	VAR jointtarget CDP_979 := [[-11.91, 35.75, 6.26, 0, 47.99, -88.67], [9E9, 9E9, 9E9, 9E9, 9E9, 9E9]];
	VAR jointtarget CDP_980 := [[-11.89, 35.75, 6.26, 0, 47.99, -88.98], [9E9, 9E9, 9E9, 9E9, 9E9, 9E9]];
	VAR jointtarget CDP_981 := [[-11.87, 35.75, 6.26, 0, 47.99, -89.63], [9E9, 9E9, 9E9, 9E9, 9E9, 9E9]];
	VAR jointtarget CDP_982 := [[-11.86, 35.75, 6.26, 0, 47.99, -90.27], [9E9, 9E9, 9E9, 9E9, 9E9, 9E9]];
	VAR jointtarget CDP_983 := [[-11.84, 35.75, 6.26, 0, 47.99, -90.92], [9E9, 9E9, 9E9, 9E9, 9E9, 9E9]];
	VAR jointtarget CDP_984 := [[-11.82, 35.75, 6.26, 0, 47.99, -91.56], [9E9, 9E9, 9E9, 9E9, 9E9, 9E9]];
	VAR jointtarget CDP_985 := [[-11.81, 35.75, 6.26, 0, 47.99, -92.21], [9E9, 9E9, 9E9, 9E9, 9E9, 9E9]];
	VAR jointtarget CDP_986 := [[-11.79, 35.75, 6.26, 0, 47.99, -92.85], [9E9, 9E9, 9E9, 9E9, 9E9, 9E9]];
	VAR jointtarget CDP_987 := [[-11.77, 35.75, 6.26, 0, 47.99, -93.5], [9E9, 9E9, 9E9, 9E9, 9E9, 9E9]];
	VAR jointtarget CDP_988 := [[-11.76, 35.75, 6.27, 0, 47.99, -94.14], [9E9, 9E9, 9E9, 9E9, 9E9, 9E9]];
	VAR jointtarget CDP_989 := [[-11.74, 35.74, 6.27, 0, 47.99, -94.79], [9E9, 9E9, 9E9, 9E9, 9E9, 9E9]];
	VAR jointtarget CDP_990 := [[-11.72, 35.74, 6.27, 0, 47.99, -95.43], [9E9, 9E9, 9E9, 9E9, 9E9, 9E9]];
	VAR jointtarget CDP_991 := [[-11.71, 35.74, 6.28, 0, 47.98, -96.08], [9E9, 9E9, 9E9, 9E9, 9E9, 9E9]];
	VAR jointtarget CDP_992 := [[-11.69, 35.74, 6.28, 0, 47.98, -96.72], [9E9, 9E9, 9E9, 9E9, 9E9, 9E9]];
	VAR jointtarget CDP_993 := [[-11.67, 35.74, 6.28, 0, 47.98, -97.37], [9E9, 9E9, 9E9, 9E9, 9E9, 9E9]];
	VAR jointtarget CDP_994 := [[-11.66, 35.73, 6.29, 0, 47.98, -98.01], [9E9, 9E9, 9E9, 9E9, 9E9, 9E9]];
	VAR jointtarget CDP_995 := [[-11.64, 35.73, 6.29, 0, 47.98, -98.66], [9E9, 9E9, 9E9, 9E9, 9E9, 9E9]];
	VAR jointtarget CDP_996 := [[-11.62, 35.73, 6.3, 0, 47.98, -99.31], [9E9, 9E9, 9E9, 9E9, 9E9, 9E9]];
	VAR jointtarget CDP_997 := [[-11.61, 35.72, 6.3, 0, 47.97, -99.95], [9E9, 9E9, 9E9, 9E9, 9E9, 9E9]];
	VAR jointtarget CDP_998 := [[-11.59, 35.72, 6.31, 0, 47.97, -100.6], [9E9, 9E9, 9E9, 9E9, 9E9, 9E9]];
	VAR jointtarget CDP_999 := [[-11.57, 35.72, 6.31, 0, 47.97, -101.24], [9E9, 9E9, 9E9, 9E9, 9E9, 9E9]];
	VAR jointtarget CDP_1000 := [[-10.48, 35.49, 6.71, 0, 47.81, -100.48], [9E9, 9E9, 9E9, 9E9, 9E9, 9E9]];
	VAR jointtarget CDP_1001 := [[-9.38, 35.28, 7.06, 0, 47.66, -99.38], [9E9, 9E9, 9E9, 9E9, 9E9, 9E9]];
	VAR jointtarget CDP_1002 := [[-8.27, 35.1, 7.37, 0, 47.53, -98.27], [9E9, 9E9, 9E9, 9E9, 9E9, 9E9]];
	VAR jointtarget CDP_1003 := [[-7.15, 34.94, 7.64, 0, 47.42, -97.15], [9E9, 9E9, 9E9, 9E9, 9E9, 9E9]];
	VAR jointtarget CDP_1004 := [[-6.03, 34.8, 7.88, 0, 47.32, -96.03], [9E9, 9E9, 9E9, 9E9, 9E9, 9E9]];
	VAR jointtarget CDP_1005 := [[-4.9, 34.69, 8.07, 0, 47.24, -94.9], [9E9, 9E9, 9E9, 9E9, 9E9, 9E9]];
	VAR jointtarget CDP_1006 := [[-3.77, 34.6, 8.22, 0, 47.18, -93.77], [9E9, 9E9, 9E9, 9E9, 9E9, 9E9]];
	VAR jointtarget CDP_1007 := [[-2.64, 34.53, 8.33, 0, 47.13, -92.64], [9E9, 9E9, 9E9, 9E9, 9E9, 9E9]];
	VAR jointtarget CDP_1008 := [[-1.51, 34.49, 8.41, 0, 47.1, -91.51], [9E9, 9E9, 9E9, 9E9, 9E9, 9E9]];
	VAR jointtarget CDP_1009 := [[-0.37, 34.47, 8.44, 0, 47.09, -90.37], [9E9, 9E9, 9E9, 9E9, 9E9, 9E9]];
	VAR jointtarget CDP_1010 := [[0.76, 34.48, 8.43, 0, 47.09, -89.24], [9E9, 9E9, 9E9, 9E9, 9E9, 9E9]];
	VAR jointtarget CDP_1011 := [[1.9, 34.5, 8.39, 0, 47.11, -88.1], [9E9, 9E9, 9E9, 9E9, 9E9, 9E9]];
	VAR jointtarget CDP_1012 := [[3.03, 34.55, 8.3, 0, 47.15, -86.97], [9E9, 9E9, 9E9, 9E9, 9E9, 9E9]];
	VAR jointtarget CDP_1013 := [[4.16, 34.63, 8.17, 0, 47.2, -85.84], [9E9, 9E9, 9E9, 9E9, 9E9, 9E9]];
	VAR jointtarget CDP_1014 := [[5.29, 34.73, 8.01, 0, 47.27, -84.71], [9E9, 9E9, 9E9, 9E9, 9E9, 9E9]];
	VAR jointtarget CDP_1015 := [[6.42, 34.85, 7.8, 0, 47.35, -83.58], [9E9, 9E9, 9E9, 9E9, 9E9, 9E9]];
	VAR jointtarget CDP_1016 := [[7.54, 34.99, 7.55, 0, 47.45, -82.46], [9E9, 9E9, 9E9, 9E9, 9E9, 9E9]];
	VAR jointtarget CDP_1017 := [[8.65, 35.16, 7.27, 0, 47.57, -81.35], [9E9, 9E9, 9E9, 9E9, 9E9, 9E9]];
	VAR jointtarget CDP_1018 := [[9.76, 35.35, 6.94, 0, 47.71, -80.24], [9E9, 9E9, 9E9, 9E9, 9E9, 9E9]];
	VAR jointtarget CDP_1019 := [[10.86, 35.56, 6.58, 0, 47.86, -79.14], [9E9, 9E9, 9E9, 9E9, 9E9, 9E9]];
	VAR jointtarget CDP_1020 := [[10.87, 35.57, 6.57, 0, 47.86, -79.46], [9E9, 9E9, 9E9, 9E9, 9E9, 9E9]];
	VAR jointtarget CDP_1021 := [[10.89, 35.57, 6.56, 0, 47.86, -80.1], [9E9, 9E9, 9E9, 9E9, 9E9, 9E9]];
	VAR jointtarget CDP_1022 := [[10.91, 35.57, 6.56, 0, 47.87, -80.75], [9E9, 9E9, 9E9, 9E9, 9E9, 9E9]];
	VAR jointtarget CDP_1023 := [[10.92, 35.58, 6.55, 0, 47.87, -81.39], [9E9, 9E9, 9E9, 9E9, 9E9, 9E9]];
	VAR jointtarget CDP_1024 := [[10.94, 35.58, 6.55, 0, 47.87, -82.04], [9E9, 9E9, 9E9, 9E9, 9E9, 9E9]];
	VAR jointtarget CDP_1025 := [[10.96, 35.58, 6.55, 0, 47.87, -82.68], [9E9, 9E9, 9E9, 9E9, 9E9, 9E9]];
	VAR jointtarget CDP_1026 := [[10.97, 35.58, 6.54, 0, 47.87, -83.33], [9E9, 9E9, 9E9, 9E9, 9E9, 9E9]];
	VAR jointtarget CDP_1027 := [[10.99, 35.59, 6.54, 0, 47.87, -83.97], [9E9, 9E9, 9E9, 9E9, 9E9, 9E9]];
	VAR jointtarget CDP_1028 := [[11.01, 35.59, 6.54, 0, 47.88, -84.62], [9E9, 9E9, 9E9, 9E9, 9E9, 9E9]];
	VAR jointtarget CDP_1029 := [[11.02, 35.59, 6.53, 0, 47.88, -85.27], [9E9, 9E9, 9E9, 9E9, 9E9, 9E9]];
	VAR jointtarget CDP_1030 := [[11.04, 35.59, 6.53, 0, 47.88, -85.91], [9E9, 9E9, 9E9, 9E9, 9E9, 9E9]];
	VAR jointtarget CDP_1031 := [[11.06, 35.59, 6.53, 0, 47.88, -86.56], [9E9, 9E9, 9E9, 9E9, 9E9, 9E9]];
	VAR jointtarget CDP_1032 := [[11.07, 35.59, 6.53, 0, 47.88, -87.2], [9E9, 9E9, 9E9, 9E9, 9E9, 9E9]];
	VAR jointtarget CDP_1033 := [[11.09, 35.59, 6.53, 0, 47.88, -87.85], [9E9, 9E9, 9E9, 9E9, 9E9, 9E9]];
	VAR jointtarget CDP_1034 := [[11.11, 35.59, 6.53, 0, 47.88, -88.49], [9E9, 9E9, 9E9, 9E9, 9E9, 9E9]];
	VAR jointtarget CDP_1035 := [[11.13, 35.59, 6.53, 0, 47.88, -89.14], [9E9, 9E9, 9E9, 9E9, 9E9, 9E9]];
	VAR jointtarget CDP_1036 := [[11.14, 35.59, 6.53, 0, 47.88, -89.78], [9E9, 9E9, 9E9, 9E9, 9E9, 9E9]];
	VAR jointtarget CDP_1037 := [[11.16, 35.59, 6.53, 0, 47.88, -90.43], [9E9, 9E9, 9E9, 9E9, 9E9, 9E9]];
	VAR jointtarget CDP_1038 := [[11.18, 35.59, 6.53, 0, 47.88, -91.07], [9E9, 9E9, 9E9, 9E9, 9E9, 9E9]];
	VAR jointtarget CDP_1039 := [[11.19, 35.59, 6.53, 0, 47.88, -91.72], [9E9, 9E9, 9E9, 9E9, 9E9, 9E9]];
	VAR jointtarget CDP_1040 := [[11.26, 35.59, 6.53, 0, 47.88, -91.98], [9E9, 9E9, 9E9, 9E9, 9E9, 9E9]];
	VAR jointtarget CDP_1041 := [[11.33, 35.59, 6.54, 0, 47.88, -91.91], [9E9, 9E9, 9E9, 9E9, 9E9, 9E9]];
	VAR jointtarget CDP_1042 := [[11.4, 35.59, 6.54, 0, 47.87, -91.84], [9E9, 9E9, 9E9, 9E9, 9E9, 9E9]];
	VAR jointtarget CDP_1043 := [[11.47, 35.58, 6.54, 0, 47.87, -91.78], [9E9, 9E9, 9E9, 9E9, 9E9, 9E9]];
	VAR jointtarget CDP_1044 := [[11.53, 35.58, 6.55, 0, 47.87, -91.71], [9E9, 9E9, 9E9, 9E9, 9E9, 9E9]];
	VAR jointtarget CDP_1045 := [[11.6, 35.58, 6.55, 0, 47.87, -91.64], [9E9, 9E9, 9E9, 9E9, 9E9, 9E9]];
	VAR jointtarget CDP_1046 := [[11.67, 35.58, 6.56, 0, 47.87, -91.57], [9E9, 9E9, 9E9, 9E9, 9E9, 9E9]];
	VAR jointtarget CDP_1047 := [[11.74, 35.57, 6.56, 0, 47.87, -91.5], [9E9, 9E9, 9E9, 9E9, 9E9, 9E9]];
	VAR jointtarget CDP_1048 := [[11.81, 35.57, 6.56, 0, 47.87, -91.44], [9E9, 9E9, 9E9, 9E9, 9E9, 9E9]];
	VAR jointtarget CDP_1049 := [[11.87, 35.57, 6.56, 0, 47.86, -91.37], [9E9, 9E9, 9E9, 9E9, 9E9, 9E9]];
	VAR jointtarget CDP_1050 := [[11.94, 35.57, 6.57, 0, 47.86, -91.3], [9E9, 9E9, 9E9, 9E9, 9E9, 9E9]];
	VAR jointtarget CDP_1051 := [[12.01, 35.57, 6.57, 0, 47.86, -91.23], [9E9, 9E9, 9E9, 9E9, 9E9, 9E9]];
	VAR jointtarget CDP_1052 := [[12.08, 35.57, 6.57, 0, 47.86, -91.16], [9E9, 9E9, 9E9, 9E9, 9E9, 9E9]];
	VAR jointtarget CDP_1053 := [[12.15, 35.56, 6.58, 0, 47.86, -91.09], [9E9, 9E9, 9E9, 9E9, 9E9, 9E9]];
	VAR jointtarget CDP_1054 := [[12.21, 35.56, 6.58, 0, 47.86, -91.03], [9E9, 9E9, 9E9, 9E9, 9E9, 9E9]];
	VAR jointtarget CDP_1055 := [[12.28, 35.56, 6.58, 0, 47.86, -90.96], [9E9, 9E9, 9E9, 9E9, 9E9, 9E9]];
	VAR jointtarget CDP_1056 := [[12.35, 35.56, 6.58, 0, 47.86, -90.89], [9E9, 9E9, 9E9, 9E9, 9E9, 9E9]];
	VAR jointtarget CDP_1057 := [[12.42, 35.56, 6.58, 0, 47.86, -90.82], [9E9, 9E9, 9E9, 9E9, 9E9, 9E9]];
	VAR jointtarget CDP_1058 := [[12.49, 35.56, 6.59, 0, 47.86, -90.75], [9E9, 9E9, 9E9, 9E9, 9E9, 9E9]];
	VAR jointtarget CDP_1059 := [[12.55, 35.56, 6.59, 0, 47.86, -90.69], [9E9, 9E9, 9E9, 9E9, 9E9, 9E9]];
	VAR jointtarget CDP_1060 := [[12.69, 35.57, 6.57, 0, 47.86, -85.39], [9E9, 9E9, 9E9, 9E9, 9E9, 9E9]];
	VAR jointtarget CDP_1061 := [[12.81, 35.61, 6.51, 0, 47.89, -74.94], [9E9, 9E9, 9E9, 9E9, 9E9, 9E9]];
	VAR jointtarget CDP_1062 := [[12.93, 35.67, 6.4, 0, 47.93, -64.5], [9E9, 9E9, 9E9, 9E9, 9E9, 9E9]];
	VAR jointtarget CDP_1063 := [[13.04, 35.75, 6.26, 0, 47.99, -54.07], [9E9, 9E9, 9E9, 9E9, 9E9, 9E9]];
	VAR jointtarget CDP_1064 := [[13.13, 35.85, 6.08, 0, 48.07, -43.65], [9E9, 9E9, 9E9, 9E9, 9E9, 9E9]];
	VAR jointtarget CDP_1065 := [[13.2, 35.97, 5.88, 0, 48.15, -33.25], [9E9, 9E9, 9E9, 9E9, 9E9, 9E9]];
	VAR jointtarget CDP_1066 := [[13.25, 36.1, 5.65, 0, 48.24, -22.88], [9E9, 9E9, 9E9, 9E9, 9E9, 9E9]];
	VAR jointtarget CDP_1067 := [[13.28, 36.24, 5.41, 0, 48.34, -12.53], [9E9, 9E9, 9E9, 9E9, 9E9, 9E9]];
	VAR jointtarget CDP_1068 := [[13.29, 36.39, 5.17, 0, 48.45, -2.2], [9E9, 9E9, 9E9, 9E9, 9E9, 9E9]];
	VAR jointtarget CDP_1069 := [[13.27, 36.53, 4.92, 0, 48.55, 8.11], [9E9, 9E9, 9E9, 9E9, 9E9, 9E9]];
	VAR jointtarget CDP_1070 := [[13.23, 36.66, 4.69, 0, 48.65, 18.39], [9E9, 9E9, 9E9, 9E9, 9E9, 9E9]];
	VAR jointtarget CDP_1071 := [[13.17, 36.79, 4.47, 0, 48.74, 28.65], [9E9, 9E9, 9E9, 9E9, 9E9, 9E9]];
	VAR jointtarget CDP_1072 := [[13.08, 36.9, 4.28, 0, 48.82, 38.9], [9E9, 9E9, 9E9, 9E9, 9E9, 9E9]];
	VAR jointtarget CDP_1073 := [[12.99, 36.99, 4.12, 0, 48.89, 49.12], [9E9, 9E9, 9E9, 9E9, 9E9, 9E9]];
	VAR jointtarget CDP_1074 := [[12.88, 37.07, 3.99, 0, 48.94, 59.33], [9E9, 9E9, 9E9, 9E9, 9E9, 9E9]];
	VAR jointtarget CDP_1075 := [[12.75, 37.12, 3.91, 0, 48.98, 69.54], [9E9, 9E9, 9E9, 9E9, 9E9, 9E9]];
	VAR jointtarget CDP_1076 := [[12.63, 37.14, 3.86, 0, 48.99, 79.73], [9E9, 9E9, 9E9, 9E9, 9E9, 9E9]];
	VAR jointtarget CDP_1077 := [[12.5, 37.14, 3.86, 0, 48.99, 89.93], [9E9, 9E9, 9E9, 9E9, 9E9, 9E9]];
	VAR jointtarget CDP_1078 := [[12.37, 37.12, 3.91, 0, 48.98, 100.13], [9E9, 9E9, 9E9, 9E9, 9E9, 9E9]];
	VAR jointtarget CDP_1079 := [[12.25, 37.07, 3.99, 0, 48.94, 110.33], [9E9, 9E9, 9E9, 9E9, 9E9, 9E9]];
	VAR jointtarget CDP_1080 := [[12.19, 37.04, 4.05, 0, 48.92, 115.43], [9E9, 9E9, 9E9, 9E9, 9E9, 9E9]];
	VAR jointtarget CDP_1081 := [[12.13, 37, 4.1, 0, 48.89, 115.37], [9E9, 9E9, 9E9, 9E9, 9E9, 9E9]];
	VAR jointtarget CDP_1082 := [[12.07, 36.97, 4.16, 0, 48.87, 115.31], [9E9, 9E9, 9E9, 9E9, 9E9, 9E9]];
	VAR jointtarget CDP_1083 := [[12.01, 36.94, 4.21, 0, 48.85, 115.25], [9E9, 9E9, 9E9, 9E9, 9E9, 9E9]];
	VAR jointtarget CDP_1084 := [[11.95, 36.91, 4.27, 0, 48.82, 115.19], [9E9, 9E9, 9E9, 9E9, 9E9, 9E9]];
	VAR jointtarget CDP_1085 := [[11.89, 36.88, 4.32, 0, 48.8, 115.13], [9E9, 9E9, 9E9, 9E9, 9E9, 9E9]];
	VAR jointtarget CDP_1086 := [[11.83, 36.85, 4.37, 0, 48.78, 115.07], [9E9, 9E9, 9E9, 9E9, 9E9, 9E9]];
	VAR jointtarget CDP_1087 := [[11.77, 36.82, 4.43, 0, 48.76, 115.01], [9E9, 9E9, 9E9, 9E9, 9E9, 9E9]];
	VAR jointtarget CDP_1088 := [[11.71, 36.78, 4.48, 0, 48.73, 114.95], [9E9, 9E9, 9E9, 9E9, 9E9, 9E9]];
	VAR jointtarget CDP_1089 := [[11.65, 36.75, 4.54, 0, 48.71, 114.89], [9E9, 9E9, 9E9, 9E9, 9E9, 9E9]];
	VAR jointtarget CDP_1090 := [[11.59, 36.72, 4.59, 0, 48.69, 114.83], [9E9, 9E9, 9E9, 9E9, 9E9, 9E9]];
	VAR jointtarget CDP_1091 := [[11.53, 36.69, 4.64, 0, 48.67, 114.77], [9E9, 9E9, 9E9, 9E9, 9E9, 9E9]];
	VAR jointtarget CDP_1092 := [[11.47, 36.66, 4.7, 0, 48.64, 114.71], [9E9, 9E9, 9E9, 9E9, 9E9, 9E9]];
	VAR jointtarget CDP_1093 := [[11.4, 36.63, 4.75, 0, 48.62, 114.64], [9E9, 9E9, 9E9, 9E9, 9E9, 9E9]];
	VAR jointtarget CDP_1094 := [[11.34, 36.6, 4.8, 0, 48.6, 114.58], [9E9, 9E9, 9E9, 9E9, 9E9, 9E9]];
	VAR jointtarget CDP_1095 := [[11.28, 36.57, 4.85, 0, 48.58, 114.52], [9E9, 9E9, 9E9, 9E9, 9E9, 9E9]];
	VAR jointtarget CDP_1096 := [[11.22, 36.54, 4.91, 0, 48.56, 114.46], [9E9, 9E9, 9E9, 9E9, 9E9, 9E9]];
	VAR jointtarget CDP_1097 := [[11.16, 36.51, 4.96, 0, 48.53, 114.4], [9E9, 9E9, 9E9, 9E9, 9E9, 9E9]];
	VAR jointtarget CDP_1098 := [[11.1, 36.48, 5.01, 0, 48.51, 114.34], [9E9, 9E9, 9E9, 9E9, 9E9, 9E9]];
	VAR jointtarget CDP_1099 := [[11.04, 36.45, 5.06, 0, 48.49, 114.28], [9E9, 9E9, 9E9, 9E9, 9E9, 9E9]];
	VAR jointtarget CDP_1100 := [[11.02, 36.44, 5.08, 0, 48.49, 113.93], [9E9, 9E9, 9E9, 9E9, 9E9, 9E9]];
	VAR jointtarget CDP_1101 := [[11.01, 36.43, 5.09, 0, 48.48, 113.26], [9E9, 9E9, 9E9, 9E9, 9E9, 9E9]];
	VAR jointtarget CDP_1102 := [[10.99, 36.43, 5.1, 0, 48.47, 112.58], [9E9, 9E9, 9E9, 9E9, 9E9, 9E9]];
	VAR jointtarget CDP_1103 := [[10.98, 36.42, 5.11, 0, 48.47, 111.9], [9E9, 9E9, 9E9, 9E9, 9E9, 9E9]];
	VAR jointtarget CDP_1104 := [[10.96, 36.41, 5.12, 0, 48.47, 111.22], [9E9, 9E9, 9E9, 9E9, 9E9, 9E9]];
	VAR jointtarget CDP_1105 := [[10.95, 36.41, 5.13, 0, 48.46, 110.55], [9E9, 9E9, 9E9, 9E9, 9E9, 9E9]];
	VAR jointtarget CDP_1106 := [[10.93, 36.4, 5.14, 0, 48.46, 109.87], [9E9, 9E9, 9E9, 9E9, 9E9, 9E9]];
	VAR jointtarget CDP_1107 := [[10.91, 36.39, 5.16, 0, 48.45, 109.19], [9E9, 9E9, 9E9, 9E9, 9E9, 9E9]];
	VAR jointtarget CDP_1108 := [[10.9, 36.39, 5.17, 0, 48.45, 108.51], [9E9, 9E9, 9E9, 9E9, 9E9, 9E9]];
	VAR jointtarget CDP_1109 := [[10.88, 36.38, 5.17, 0, 48.44, 107.83], [9E9, 9E9, 9E9, 9E9, 9E9, 9E9]];
	VAR jointtarget CDP_1110 := [[10.87, 36.38, 5.18, 0, 48.44, 107.16], [9E9, 9E9, 9E9, 9E9, 9E9, 9E9]];
	VAR jointtarget CDP_1111 := [[10.85, 36.37, 5.19, 0, 48.44, 106.48], [9E9, 9E9, 9E9, 9E9, 9E9, 9E9]];
	VAR jointtarget CDP_1112 := [[10.83, 36.37, 5.2, 0, 48.43, 105.8], [9E9, 9E9, 9E9, 9E9, 9E9, 9E9]];
	VAR jointtarget CDP_1113 := [[10.82, 36.36, 5.21, 0, 48.43, 105.12], [9E9, 9E9, 9E9, 9E9, 9E9, 9E9]];
	VAR jointtarget CDP_1114 := [[10.8, 36.36, 5.22, 0, 48.43, 104.44], [9E9, 9E9, 9E9, 9E9, 9E9, 9E9]];
	VAR jointtarget CDP_1115 := [[10.79, 36.35, 5.22, 0, 48.42, 103.77], [9E9, 9E9, 9E9, 9E9, 9E9, 9E9]];
	VAR jointtarget CDP_1116 := [[10.77, 36.35, 5.23, 0, 48.42, 103.09], [9E9, 9E9, 9E9, 9E9, 9E9, 9E9]];
	VAR jointtarget CDP_1117 := [[10.75, 36.34, 5.24, 0, 48.42, 102.41], [9E9, 9E9, 9E9, 9E9, 9E9, 9E9]];
	VAR jointtarget CDP_1118 := [[10.74, 36.34, 5.24, 0, 48.41, 101.73], [9E9, 9E9, 9E9, 9E9, 9E9, 9E9]];
	VAR jointtarget CDP_1119 := [[10.72, 36.34, 5.25, 0, 48.41, 101.05], [9E9, 9E9, 9E9, 9E9, 9E9, 9E9]];
	VAR jointtarget CDP_1120 := [[9.64, 36.13, 5.61, 0, 48.26, 99.64], [9E9, 9E9, 9E9, 9E9, 9E9, 9E9]];
	VAR jointtarget CDP_1121 := [[8.56, 35.94, 5.94, 0, 48.13, 98.56], [9E9, 9E9, 9E9, 9E9, 9E9, 9E9]];
	VAR jointtarget CDP_1122 := [[7.47, 35.77, 6.22, 0, 48.01, 97.47], [9E9, 9E9, 9E9, 9E9, 9E9, 9E9]];
	VAR jointtarget CDP_1123 := [[6.38, 35.63, 6.46, 0, 47.91, 96.38], [9E9, 9E9, 9E9, 9E9, 9E9, 9E9]];
	VAR jointtarget CDP_1124 := [[5.28, 35.51, 6.67, 0, 47.82, 95.28], [9E9, 9E9, 9E9, 9E9, 9E9, 9E9]];
	VAR jointtarget CDP_1125 := [[4.17, 35.41, 6.84, 0, 47.75, 94.17], [9E9, 9E9, 9E9, 9E9, 9E9, 9E9]];
	VAR jointtarget CDP_1126 := [[3.07, 35.34, 6.97, 0, 47.7, 93.07], [9E9, 9E9, 9E9, 9E9, 9E9, 9E9]];
	VAR jointtarget CDP_1127 := [[1.96, 35.28, 7.05, 0, 47.66, 91.96], [9E9, 9E9, 9E9, 9E9, 9E9, 9E9]];
	VAR jointtarget CDP_1128 := [[0.85, 35.26, 7.1, 0, 47.64, 90.85], [9E9, 9E9, 9E9, 9E9, 9E9, 9E9]];
	VAR jointtarget CDP_1129 := [[-0.26, 35.25, 7.11, 0, 47.64, 89.74], [9E9, 9E9, 9E9, 9E9, 9E9, 9E9]];
	VAR jointtarget CDP_1130 := [[-1.37, 35.27, 7.08, 0, 47.65, 88.63], [9E9, 9E9, 9E9, 9E9, 9E9, 9E9]];
	VAR jointtarget CDP_1131 := [[-2.48, 35.31, 7.02, 0, 47.68, 87.52], [9E9, 9E9, 9E9, 9E9, 9E9, 9E9]];
	VAR jointtarget CDP_1132 := [[-3.59, 35.37, 6.91, 0, 47.72, 86.41], [9E9, 9E9, 9E9, 9E9, 9E9, 9E9]];
	VAR jointtarget CDP_1133 := [[-4.7, 35.45, 6.76, 0, 47.78, 85.3], [9E9, 9E9, 9E9, 9E9, 9E9, 9E9]];
	VAR jointtarget CDP_1134 := [[-5.8, 35.56, 6.58, 0, 47.86, 84.2], [9E9, 9E9, 9E9, 9E9, 9E9, 9E9]];
	VAR jointtarget CDP_1135 := [[-6.9, 35.69, 6.35, 0, 47.95, 83.1], [9E9, 9E9, 9E9, 9E9, 9E9, 9E9]];
	VAR jointtarget CDP_1136 := [[-7.99, 35.85, 6.09, 0, 48.06, 82.01], [9E9, 9E9, 9E9, 9E9, 9E9, 9E9]];
	VAR jointtarget CDP_1137 := [[-9.08, 36.02, 5.79, 0, 48.19, 80.92], [9E9, 9E9, 9E9, 9E9, 9E9, 9E9]];
	VAR jointtarget CDP_1138 := [[-10.16, 36.22, 5.45, 0, 48.33, 79.84], [9E9, 9E9, 9E9, 9E9, 9E9, 9E9]];
	VAR jointtarget CDP_1139 := [[-11.23, 36.45, 5.07, 0, 48.49, 78.77], [9E9, 9E9, 9E9, 9E9, 9E9, 9E9]];
	VAR jointtarget CDP_1140 := [[-11.28, 36.46, 5.05, 0, 48.5, 79.81], [9E9, 9E9, 9E9, 9E9, 9E9, 9E9]];
	VAR jointtarget CDP_1141 := [[-11.34, 36.46, 5.03, 0, 48.5, 81.95], [9E9, 9E9, 9E9, 9E9, 9E9, 9E9]];
	VAR jointtarget CDP_1142 := [[-11.39, 36.47, 5.02, 0, 48.51, 84.09], [9E9, 9E9, 9E9, 9E9, 9E9, 9E9]];
	VAR jointtarget CDP_1143 := [[-11.45, 36.47, 5.02, 0, 48.51, 86.23], [9E9, 9E9, 9E9, 9E9, 9E9, 9E9]];
	VAR jointtarget CDP_1144 := [[-11.5, 36.48, 5.01, 0, 48.51, 88.37], [9E9, 9E9, 9E9, 9E9, 9E9, 9E9]];
	VAR jointtarget CDP_1145 := [[-11.56, 36.48, 5.01, 0, 48.51, 90.51], [9E9, 9E9, 9E9, 9E9, 9E9, 9E9]];
	VAR jointtarget CDP_1146 := [[-11.61, 36.47, 5.02, 0, 48.51, 92.65], [9E9, 9E9, 9E9, 9E9, 9E9, 9E9]];
	VAR jointtarget CDP_1147 := [[-11.67, 36.47, 5.03, 0, 48.51, 94.78], [9E9, 9E9, 9E9, 9E9, 9E9, 9E9]];
	VAR jointtarget CDP_1148 := [[-11.72, 36.46, 5.04, 0, 48.5, 96.92], [9E9, 9E9, 9E9, 9E9, 9E9, 9E9]];
	VAR jointtarget CDP_1149 := [[-11.78, 36.45, 5.06, 0, 48.49, 99.06], [9E9, 9E9, 9E9, 9E9, 9E9, 9E9]];
	VAR jointtarget CDP_1150 := [[-11.83, 36.44, 5.08, 0, 48.48, 101.2], [9E9, 9E9, 9E9, 9E9, 9E9, 9E9]];
	VAR jointtarget CDP_1151 := [[-11.89, 36.43, 5.1, 0, 48.47, 103.34], [9E9, 9E9, 9E9, 9E9, 9E9, 9E9]];
	VAR jointtarget CDP_1152 := [[-11.94, 36.41, 5.13, 0, 48.46, 105.48], [9E9, 9E9, 9E9, 9E9, 9E9, 9E9]];
	VAR jointtarget CDP_1153 := [[-11.99, 36.39, 5.16, 0, 48.45, 107.63], [9E9, 9E9, 9E9, 9E9, 9E9, 9E9]];
	VAR jointtarget CDP_1154 := [[-12.04, 36.37, 5.19, 0, 48.44, 109.77], [9E9, 9E9, 9E9, 9E9, 9E9, 9E9]];
	VAR jointtarget CDP_1155 := [[-12.09, 36.35, 5.23, 0, 48.42, 111.91], [9E9, 9E9, 9E9, 9E9, 9E9, 9E9]];
	VAR jointtarget CDP_1156 := [[-12.15, 36.32, 5.28, 0, 48.4, 114.05], [9E9, 9E9, 9E9, 9E9, 9E9, 9E9]];
	VAR jointtarget CDP_1157 := [[-12.19, 36.3, 5.32, 0, 48.38, 116.2], [9E9, 9E9, 9E9, 9E9, 9E9, 9E9]];
	VAR jointtarget CDP_1158 := [[-12.24, 36.27, 5.37, 0, 48.36, 118.34], [9E9, 9E9, 9E9, 9E9, 9E9, 9E9]];
	VAR jointtarget CDP_1159 := [[-12.29, 36.24, 5.42, 0, 48.34, 120.49], [9E9, 9E9, 9E9, 9E9, 9E9, 9E9]];
	VAR jointtarget CDP_1160 := [[-12.32, 36.22, 5.46, 0, 48.33, 121.56], [9E9, 9E9, 9E9, 9E9, 9E9, 9E9]];
	VAR jointtarget CDP_1161 := [[-12.35, 36.2, 5.49, 0, 48.31, 121.53], [9E9, 9E9, 9E9, 9E9, 9E9, 9E9]];
	VAR jointtarget CDP_1162 := [[-12.38, 36.18, 5.52, 0, 48.3, 121.5], [9E9, 9E9, 9E9, 9E9, 9E9, 9E9]];
	VAR jointtarget CDP_1163 := [[-12.41, 36.16, 5.55, 0, 48.29, 121.47], [9E9, 9E9, 9E9, 9E9, 9E9, 9E9]];
	VAR jointtarget CDP_1164 := [[-12.43, 36.14, 5.59, 0, 48.27, 121.44], [9E9, 9E9, 9E9, 9E9, 9E9, 9E9]];
	VAR jointtarget CDP_1165 := [[-12.46, 36.12, 5.62, 0, 48.26, 121.41], [9E9, 9E9, 9E9, 9E9, 9E9, 9E9]];
	VAR jointtarget CDP_1166 := [[-12.49, 36.1, 5.65, 0, 48.24, 121.39], [9E9, 9E9, 9E9, 9E9, 9E9, 9E9]];
	VAR jointtarget CDP_1167 := [[-12.52, 36.08, 5.68, 0, 48.23, 121.36], [9E9, 9E9, 9E9, 9E9, 9E9, 9E9]];
	VAR jointtarget CDP_1168 := [[-12.55, 36.07, 5.72, 0, 48.22, 121.33], [9E9, 9E9, 9E9, 9E9, 9E9, 9E9]];
	VAR jointtarget CDP_1169 := [[-12.58, 36.05, 5.75, 0, 48.2, 121.3], [9E9, 9E9, 9E9, 9E9, 9E9, 9E9]];
	VAR jointtarget CDP_1170 := [[-12.61, 36.03, 5.78, 0, 48.19, 121.27], [9E9, 9E9, 9E9, 9E9, 9E9, 9E9]];
	VAR jointtarget CDP_1171 := [[-12.63, 36.01, 5.81, 0, 48.18, 121.24], [9E9, 9E9, 9E9, 9E9, 9E9, 9E9]];
	VAR jointtarget CDP_1172 := [[-12.66, 35.99, 5.85, 0, 48.16, 121.21], [9E9, 9E9, 9E9, 9E9, 9E9, 9E9]];
	VAR jointtarget CDP_1173 := [[-12.69, 35.97, 5.88, 0, 48.15, 121.18], [9E9, 9E9, 9E9, 9E9, 9E9, 9E9]];
	VAR jointtarget CDP_1174 := [[-12.72, 35.95, 5.91, 0, 48.14, 121.16], [9E9, 9E9, 9E9, 9E9, 9E9, 9E9]];
	VAR jointtarget CDP_1175 := [[-12.75, 35.93, 5.94, 0, 48.12, 121.13], [9E9, 9E9, 9E9, 9E9, 9E9, 9E9]];
	VAR jointtarget CDP_1176 := [[-12.78, 35.91, 5.98, 0, 48.11, 121.1], [9E9, 9E9, 9E9, 9E9, 9E9, 9E9]];
	VAR jointtarget CDP_1177 := [[-12.81, 35.9, 6.01, 0, 48.1, 121.07], [9E9, 9E9, 9E9, 9E9, 9E9, 9E9]];
	VAR jointtarget CDP_1178 := [[-12.84, 35.88, 6.04, 0, 48.08, 121.04], [9E9, 9E9, 9E9, 9E9, 9E9, 9E9]];
	VAR jointtarget CDP_1179 := [[-12.86, 35.86, 6.07, 0, 48.07, 121.01], [9E9, 9E9, 9E9, 9E9, 9E9, 9E9]];
	VAR jointtarget CDP_1180 := [[-13.02, 35.79, 6.2, 0, 48.02, 114.17], [9E9, 9E9, 9E9, 9E9, 9E9, 9E9]];
	VAR jointtarget CDP_1181 := [[-13.18, 35.75, 6.25, 0, 47.99, 100.62], [9E9, 9E9, 9E9, 9E9, 9E9, 9E9]];
	VAR jointtarget CDP_1182 := [[-13.34, 35.76, 6.24, 0, 48, 87.07], [9E9, 9E9, 9E9, 9E9, 9E9, 9E9]];
	VAR jointtarget CDP_1183 := [[-13.5, 35.81, 6.15, 0, 48.04, 73.52], [9E9, 9E9, 9E9, 9E9, 9E9, 9E9]];
	VAR jointtarget CDP_1184 := [[-13.64, 35.9, 6, 0, 48.1, 59.99], [9E9, 9E9, 9E9, 9E9, 9E9, 9E9]];
	VAR jointtarget CDP_1185 := [[-13.76, 36.02, 5.79, 0, 48.19, 46.48], [9E9, 9E9, 9E9, 9E9, 9E9, 9E9]];
	VAR jointtarget CDP_1186 := [[-13.85, 36.17, 5.53, 0, 48.29, 33.01], [9E9, 9E9, 9E9, 9E9, 9E9, 9E9]];
	VAR jointtarget CDP_1187 := [[-13.91, 36.34, 5.25, 0, 48.41, 19.56], [9E9, 9E9, 9E9, 9E9, 9E9, 9E9]];
	VAR jointtarget CDP_1188 := [[-13.92, 36.52, 4.94, 0, 48.54, 6.16], [9E9, 9E9, 9E9, 9E9, 9E9, 9E9]];
	VAR jointtarget CDP_1189 := [[-13.9, 36.7, 4.63, 0, 48.67, -7.21], [9E9, 9E9, 9E9, 9E9, 9E9, 9E9]];
	VAR jointtarget CDP_1190 := [[-13.85, 36.86, 4.35, 0, 48.79, -20.54], [9E9, 9E9, 9E9, 9E9, 9E9, 9E9]];
	VAR jointtarget CDP_1191 := [[-13.76, 37.01, 4.09, 0, 48.9, -33.84], [9E9, 9E9, 9E9, 9E9, 9E9, 9E9]];
	VAR jointtarget CDP_1192 := [[-13.64, 37.13, 3.88, 0, 48.99, -47.11], [9E9, 9E9, 9E9, 9E9, 9E9, 9E9]];
	VAR jointtarget CDP_1193 := [[-13.5, 37.22, 3.72, 0, 49.05, -60.35], [9E9, 9E9, 9E9, 9E9, 9E9, 9E9]];
	VAR jointtarget CDP_1194 := [[-13.34, 37.27, 3.64, 0, 49.09, -73.59], [9E9, 9E9, 9E9, 9E9, 9E9, 9E9]];
	VAR jointtarget CDP_1195 := [[-13.18, 37.28, 3.62, 0, 49.1, -86.81], [9E9, 9E9, 9E9, 9E9, 9E9, 9E9]];
	VAR jointtarget CDP_1196 := [[-13.02, 37.25, 3.68, 0, 49.07, -100.04], [9E9, 9E9, 9E9, 9E9, 9E9, 9E9]];
	VAR jointtarget CDP_1197 := [[-12.88, 37.18, 3.8, 0, 49.02, -113.28], [9E9, 9E9, 9E9, 9E9, 9E9, 9E9]];
	VAR jointtarget CDP_1198 := [[-12.75, 37.07, 3.98, 0, 48.94, -126.54], [9E9, 9E9, 9E9, 9E9, 9E9, 9E9]];
	VAR jointtarget CDP_1199 := [[-12.64, 36.94, 4.22, 0, 48.84, -139.82], [9E9, 9E9, 9E9, 9E9, 9E9, 9E9]];
	VAR jointtarget CDP_1200 := [[-12.62, 36.89, 4.29, 0, 48.81, -146.49], [9E9, 9E9, 9E9, 9E9, 9E9, 9E9]];
	VAR jointtarget CDP_1201 := [[-12.59, 36.85, 4.36, 0, 48.78, -146.47], [9E9, 9E9, 9E9, 9E9, 9E9, 9E9]];
	VAR jointtarget CDP_1202 := [[-12.57, 36.81, 4.43, 0, 48.75, -146.44], [9E9, 9E9, 9E9, 9E9, 9E9, 9E9]];
	VAR jointtarget CDP_1203 := [[-12.54, 36.77, 4.5, 0, 48.72, -146.42], [9E9, 9E9, 9E9, 9E9, 9E9, 9E9]];
	VAR jointtarget CDP_1204 := [[-12.52, 36.73, 4.57, 0, 48.69, -146.4], [9E9, 9E9, 9E9, 9E9, 9E9, 9E9]];
	VAR jointtarget CDP_1205 := [[-12.49, 36.69, 4.65, 0, 48.67, -146.37], [9E9, 9E9, 9E9, 9E9, 9E9, 9E9]];
	VAR jointtarget CDP_1206 := [[-12.47, 36.65, 4.72, 0, 48.64, -146.35], [9E9, 9E9, 9E9, 9E9, 9E9, 9E9]];
	VAR jointtarget CDP_1207 := [[-12.44, 36.61, 4.79, 0, 48.61, -146.32], [9E9, 9E9, 9E9, 9E9, 9E9, 9E9]];
	VAR jointtarget CDP_1208 := [[-12.42, 36.57, 4.86, 0, 48.58, -146.3], [9E9, 9E9, 9E9, 9E9, 9E9, 9E9]];
	VAR jointtarget CDP_1209 := [[-12.39, 36.53, 4.93, 0, 48.55, -146.27], [9E9, 9E9, 9E9, 9E9, 9E9, 9E9]];
	VAR jointtarget CDP_1210 := [[-12.37, 36.48, 5, 0, 48.52, -146.25], [9E9, 9E9, 9E9, 9E9, 9E9, 9E9]];
	VAR jointtarget CDP_1211 := [[-12.34, 36.44, 5.07, 0, 48.49, -146.22], [9E9, 9E9, 9E9, 9E9, 9E9, 9E9]];
	VAR jointtarget CDP_1212 := [[-12.32, 36.4, 5.14, 0, 48.46, -146.2], [9E9, 9E9, 9E9, 9E9, 9E9, 9E9]];
	VAR jointtarget CDP_1213 := [[-12.29, 36.36, 5.21, 0, 48.43, -146.17], [9E9, 9E9, 9E9, 9E9, 9E9, 9E9]];
	VAR jointtarget CDP_1214 := [[-12.27, 36.32, 5.28, 0, 48.4, -146.15], [9E9, 9E9, 9E9, 9E9, 9E9, 9E9]];
	VAR jointtarget CDP_1215 := [[-12.24, 36.28, 5.35, 0, 48.37, -146.12], [9E9, 9E9, 9E9, 9E9, 9E9, 9E9]];
	VAR jointtarget CDP_1216 := [[-12.22, 36.24, 5.42, 0, 48.34, -146.1], [9E9, 9E9, 9E9, 9E9, 9E9, 9E9]];
	VAR jointtarget CDP_1217 := [[-12.19, 36.2, 5.49, 0, 48.31, -146.07], [9E9, 9E9, 9E9, 9E9, 9E9, 9E9]];
	VAR jointtarget CDP_1218 := [[-12.17, 36.16, 5.56, 0, 48.28, -146.05], [9E9, 9E9, 9E9, 9E9, 9E9, 9E9]];
	VAR jointtarget CDP_1219 := [[-12.14, 36.12, 5.63, 0, 48.25, -146.02], [9E9, 9E9, 9E9, 9E9, 9E9, 9E9]];
	VAR jointtarget CDP_1220 := [[-12.14, 36.1, 5.65, 0, 48.24, -145.46], [9E9, 9E9, 9E9, 9E9, 9E9, 9E9]];
	VAR jointtarget CDP_1221 := [[-12.13, 36.09, 5.67, 0, 48.24, -144.35], [9E9, 9E9, 9E9, 9E9, 9E9, 9E9]];
	VAR jointtarget CDP_1222 := [[-12.12, 36.08, 5.69, 0, 48.23, -143.24], [9E9, 9E9, 9E9, 9E9, 9E9, 9E9]];
	VAR jointtarget CDP_1223 := [[-12.11, 36.07, 5.71, 0, 48.22, -142.13], [9E9, 9E9, 9E9, 9E9, 9E9, 9E9]];
	VAR jointtarget CDP_1224 := [[-12.1, 36.06, 5.73, 0, 48.21, -141.01], [9E9, 9E9, 9E9, 9E9, 9E9, 9E9]];
	VAR jointtarget CDP_1225 := [[-12.09, 36.04, 5.75, 0, 48.2, -139.9], [9E9, 9E9, 9E9, 9E9, 9E9, 9E9]];
	VAR jointtarget CDP_1226 := [[-12.08, 36.03, 5.77, 0, 48.19, -138.79], [9E9, 9E9, 9E9, 9E9, 9E9, 9E9]];
	VAR jointtarget CDP_1227 := [[-12.07, 36.02, 5.79, 0, 48.19, -137.68], [9E9, 9E9, 9E9, 9E9, 9E9, 9E9]];
	VAR jointtarget CDP_1228 := [[-12.06, 36.01, 5.81, 0, 48.18, -136.56], [9E9, 9E9, 9E9, 9E9, 9E9, 9E9]];
	VAR jointtarget CDP_1229 := [[-12.05, 36, 5.83, 0, 48.17, -135.45], [9E9, 9E9, 9E9, 9E9, 9E9, 9E9]];
	VAR jointtarget CDP_1230 := [[-12.04, 35.99, 5.85, 0, 48.16, -134.34], [9E9, 9E9, 9E9, 9E9, 9E9, 9E9]];
	VAR jointtarget CDP_1231 := [[-12.03, 35.98, 5.87, 0, 48.16, -133.22], [9E9, 9E9, 9E9, 9E9, 9E9, 9E9]];
	VAR jointtarget CDP_1232 := [[-12.02, 35.97, 5.88, 0, 48.15, -132.11], [9E9, 9E9, 9E9, 9E9, 9E9, 9E9]];
	VAR jointtarget CDP_1233 := [[-12.01, 35.96, 5.9, 0, 48.14, -130.99], [9E9, 9E9, 9E9, 9E9, 9E9, 9E9]];
	VAR jointtarget CDP_1234 := [[-12, 35.95, 5.92, 0, 48.14, -129.88], [9E9, 9E9, 9E9, 9E9, 9E9, 9E9]];
	VAR jointtarget CDP_1235 := [[-11.99, 35.94, 5.93, 0, 48.13, -128.76], [9E9, 9E9, 9E9, 9E9, 9E9, 9E9]];
	VAR jointtarget CDP_1236 := [[-11.98, 35.93, 5.95, 0, 48.12, -127.65], [9E9, 9E9, 9E9, 9E9, 9E9, 9E9]];
	VAR jointtarget CDP_1237 := [[-11.97, 35.92, 5.97, 0, 48.12, -126.53], [9E9, 9E9, 9E9, 9E9, 9E9, 9E9]];
	VAR jointtarget CDP_1238 := [[-11.96, 35.91, 5.98, 0, 48.11, -125.42], [9E9, 9E9, 9E9, 9E9, 9E9, 9E9]];
	VAR jointtarget CDP_1239 := [[-11.95, 35.9, 5.99, 0, 48.11, -124.3], [9E9, 9E9, 9E9, 9E9, 9E9, 9E9]];
	VAR jointtarget CDP_1240 := [[-11.94, 35.89, 6.01, 0, 48.1, -123.74], [9E9, 9E9, 9E9, 9E9, 9E9, 9E9]];
	VAR jointtarget CDP_1241 := [[-11.93, 35.88, 6.02, 0, 48.1, -123.73], [9E9, 9E9, 9E9, 9E9, 9E9, 9E9]];
	VAR jointtarget CDP_1242 := [[-11.92, 35.87, 6.03, 0, 48.09, -123.72], [9E9, 9E9, 9E9, 9E9, 9E9, 9E9]];
	VAR jointtarget CDP_1243 := [[-11.9, 35.87, 6.05, 0, 48.09, -123.71], [9E9, 9E9, 9E9, 9E9, 9E9, 9E9]];
	VAR jointtarget CDP_1244 := [[-11.89, 35.86, 6.06, 0, 48.08, -123.7], [9E9, 9E9, 9E9, 9E9, 9E9, 9E9]];
	VAR jointtarget CDP_1245 := [[-11.88, 35.85, 6.07, 0, 48.08, -123.69], [9E9, 9E9, 9E9, 9E9, 9E9, 9E9]];
	VAR jointtarget CDP_1246 := [[-11.87, 35.84, 6.08, 0, 48.07, -123.68], [9E9, 9E9, 9E9, 9E9, 9E9, 9E9]];
	VAR jointtarget CDP_1247 := [[-11.86, 35.84, 6.1, 0, 48.07, -123.66], [9E9, 9E9, 9E9, 9E9, 9E9, 9E9]];
	VAR jointtarget CDP_1248 := [[-11.85, 35.83, 6.11, 0, 48.06, -123.65], [9E9, 9E9, 9E9, 9E9, 9E9, 9E9]];
	VAR jointtarget CDP_1249 := [[-11.84, 35.82, 6.12, 0, 48.06, -123.64], [9E9, 9E9, 9E9, 9E9, 9E9, 9E9]];
	VAR jointtarget CDP_1250 := [[-11.83, 35.81, 6.13, 0, 48.05, -123.63], [9E9, 9E9, 9E9, 9E9, 9E9, 9E9]];
	VAR jointtarget CDP_1251 := [[-11.82, 35.8, 6.15, 0, 48.05, -123.62], [9E9, 9E9, 9E9, 9E9, 9E9, 9E9]];
	VAR jointtarget CDP_1252 := [[-11.81, 35.8, 6.16, 0, 48.04, -123.61], [9E9, 9E9, 9E9, 9E9, 9E9, 9E9]];
	VAR jointtarget CDP_1253 := [[-11.8, 35.79, 6.17, 0, 48.04, -123.6], [9E9, 9E9, 9E9, 9E9, 9E9, 9E9]];
	VAR jointtarget CDP_1254 := [[-11.79, 35.78, 6.19, 0, 48.03, -123.59], [9E9, 9E9, 9E9, 9E9, 9E9, 9E9]];
	VAR jointtarget CDP_1255 := [[-11.78, 35.77, 6.2, 0, 48.03, -123.58], [9E9, 9E9, 9E9, 9E9, 9E9, 9E9]];
	VAR jointtarget CDP_1256 := [[-11.77, 35.76, 6.21, 0, 48.02, -123.57], [9E9, 9E9, 9E9, 9E9, 9E9, 9E9]];
	VAR jointtarget CDP_1257 := [[-11.76, 35.76, 6.22, 0, 48.02, -123.56], [9E9, 9E9, 9E9, 9E9, 9E9, 9E9]];
	VAR jointtarget CDP_1258 := [[-11.75, 35.75, 6.24, 0, 48.02, -123.55], [9E9, 9E9, 9E9, 9E9, 9E9, 9E9]];
	VAR jointtarget CDP_1259 := [[-11.74, 35.74, 6.25, 0, 48.01, -123.54], [9E9, 9E9, 9E9, 9E9, 9E9, 9E9]];
	VAR jointtarget CDP_1260 := [[-10.65, 35.51, 6.65, 0, 47.85, -100.65], [9E9, 9E9, 9E9, 9E9, 9E9, 9E9]];
	VAR jointtarget CDP_1261 := [[-9.55, 35.3, 7, 0, 47.7, -99.55], [9E9, 9E9, 9E9, 9E9, 9E9, 9E9]];
	VAR jointtarget CDP_1262 := [[-8.44, 35.11, 7.32, 0, 47.57, -98.44], [9E9, 9E9, 9E9, 9E9, 9E9, 9E9]];
	VAR jointtarget CDP_1263 := [[-7.33, 34.95, 7.6, 0, 47.45, -97.33], [9E9, 9E9, 9E9, 9E9, 9E9, 9E9]];
	VAR jointtarget CDP_1264 := [[-6.21, 34.81, 7.84, 0, 47.35, -96.21], [9E9, 9E9, 9E9, 9E9, 9E9, 9E9]];
	VAR jointtarget CDP_1265 := [[-5.09, 34.69, 8.04, 0, 47.27, -95.09], [9E9, 9E9, 9E9, 9E9, 9E9, 9E9]];
	VAR jointtarget CDP_1266 := [[-3.96, 34.6, 8.2, 0, 47.2, -93.96], [9E9, 9E9, 9E9, 9E9, 9E9, 9E9]];
	VAR jointtarget CDP_1267 := [[-2.83, 34.53, 8.32, 0, 47.15, -92.83], [9E9, 9E9, 9E9, 9E9, 9E9, 9E9]];
	VAR jointtarget CDP_1268 := [[-1.7, 34.48, 8.4, 0, 47.12, -91.7], [9E9, 9E9, 9E9, 9E9, 9E9, 9E9]];
	VAR jointtarget CDP_1269 := [[-0.56, 34.46, 8.44, 0, 47.11, -90.56], [9E9, 9E9, 9E9, 9E9, 9E9, 9E9]];
	VAR jointtarget CDP_1270 := [[0.57, 34.46, 8.44, 0, 47.11, -89.43], [9E9, 9E9, 9E9, 9E9, 9E9, 9E9]];
	VAR jointtarget CDP_1271 := [[1.7, 34.48, 8.4, 0, 47.12, -88.3], [9E9, 9E9, 9E9, 9E9, 9E9, 9E9]];
	VAR jointtarget CDP_1272 := [[2.84, 34.53, 8.32, 0, 47.16, -87.16], [9E9, 9E9, 9E9, 9E9, 9E9, 9E9]];
	VAR jointtarget CDP_1273 := [[3.97, 34.6, 8.2, 0, 47.2, -86.03], [9E9, 9E9, 9E9, 9E9, 9E9, 9E9]];
	VAR jointtarget CDP_1274 := [[5.09, 34.69, 8.04, 0, 47.27, -84.91], [9E9, 9E9, 9E9, 9E9, 9E9, 9E9]];
	VAR jointtarget CDP_1275 := [[6.22, 34.81, 7.84, 0, 47.35, -83.78], [9E9, 9E9, 9E9, 9E9, 9E9, 9E9]];
	VAR jointtarget CDP_1276 := [[7.34, 34.95, 7.6, 0, 47.45, -82.66], [9E9, 9E9, 9E9, 9E9, 9E9, 9E9]];
	VAR jointtarget CDP_1277 := [[8.45, 35.11, 7.32, 0, 47.57, -81.55], [9E9, 9E9, 9E9, 9E9, 9E9, 9E9]];
	VAR jointtarget CDP_1278 := [[9.56, 35.3, 7, 0, 47.7, -80.44], [9E9, 9E9, 9E9, 9E9, 9E9, 9E9]];
	VAR jointtarget CDP_1279 := [[10.65, 35.51, 6.64, 0, 47.85, -79.35], [9E9, 9E9, 9E9, 9E9, 9E9, 9E9]];
	VAR jointtarget CDP_1280 := [[10.71, 35.52, 6.62, 0, 47.86, -78.19], [9E9, 9E9, 9E9, 9E9, 9E9, 9E9]];
	VAR jointtarget CDP_1281 := [[10.76, 35.54, 6.6, 0, 47.87, -75.95], [9E9, 9E9, 9E9, 9E9, 9E9, 9E9]];
	VAR jointtarget CDP_1282 := [[10.82, 35.55, 6.57, 0, 47.88, -73.7], [9E9, 9E9, 9E9, 9E9, 9E9, 9E9]];
	VAR jointtarget CDP_1283 := [[10.87, 35.57, 6.54, 0, 47.89, -71.45], [9E9, 9E9, 9E9, 9E9, 9E9, 9E9]];
	VAR jointtarget CDP_1284 := [[10.92, 35.59, 6.5, 0, 47.91, -69.2], [9E9, 9E9, 9E9, 9E9, 9E9, 9E9]];
	VAR jointtarget CDP_1285 := [[10.97, 35.62, 6.46, 0, 47.92, -66.96], [9E9, 9E9, 9E9, 9E9, 9E9, 9E9]];
	VAR jointtarget CDP_1286 := [[11.03, 35.64, 6.42, 0, 47.94, -64.72], [9E9, 9E9, 9E9, 9E9, 9E9, 9E9]];
	VAR jointtarget CDP_1287 := [[11.07, 35.67, 6.37, 0, 47.96, -62.47], [9E9, 9E9, 9E9, 9E9, 9E9, 9E9]];
	VAR jointtarget CDP_1288 := [[11.12, 35.7, 6.32, 0, 47.98, -60.23], [9E9, 9E9, 9E9, 9E9, 9E9, 9E9]];
	VAR jointtarget CDP_1289 := [[11.17, 35.73, 6.26, 0, 48, -57.99], [9E9, 9E9, 9E9, 9E9, 9E9, 9E9]];
	VAR jointtarget CDP_1290 := [[11.22, 35.77, 6.2, 0, 48.03, -55.75], [9E9, 9E9, 9E9, 9E9, 9E9, 9E9]];
	VAR jointtarget CDP_1291 := [[11.26, 35.8, 6.14, 0, 48.05, -53.51], [9E9, 9E9, 9E9, 9E9, 9E9, 9E9]];
	VAR jointtarget CDP_1292 := [[11.3, 35.84, 6.08, 0, 48.08, -51.27], [9E9, 9E9, 9E9, 9E9, 9E9, 9E9]];
	VAR jointtarget CDP_1293 := [[11.35, 35.88, 6.01, 0, 48.11, -49.04], [9E9, 9E9, 9E9, 9E9, 9E9, 9E9]];
	VAR jointtarget CDP_1294 := [[11.39, 35.92, 5.94, 0, 48.14, -46.8], [9E9, 9E9, 9E9, 9E9, 9E9, 9E9]];
	VAR jointtarget CDP_1295 := [[11.43, 35.96, 5.87, 0, 48.17, -44.57], [9E9, 9E9, 9E9, 9E9, 9E9, 9E9]];
	VAR jointtarget CDP_1296 := [[11.46, 36.01, 5.79, 0, 48.2, -42.34], [9E9, 9E9, 9E9, 9E9, 9E9, 9E9]];
	VAR jointtarget CDP_1297 := [[11.5, 36.05, 5.71, 0, 48.23, -40.11], [9E9, 9E9, 9E9, 9E9, 9E9, 9E9]];
	VAR jointtarget CDP_1298 := [[11.53, 36.1, 5.63, 0, 48.27, -37.88], [9E9, 9E9, 9E9, 9E9, 9E9, 9E9]];
	VAR jointtarget CDP_1299 := [[11.57, 36.15, 5.55, 0, 48.3, -35.65], [9E9, 9E9, 9E9, 9E9, 9E9, 9E9]];
	VAR jointtarget CDP_1300 := [[11.59, 36.18, 5.49, 0, 48.32, -34.54], [9E9, 9E9, 9E9, 9E9, 9E9, 9E9]];
	VAR jointtarget CDP_1301 := [[11.6, 36.21, 5.44, 0, 48.35, -34.52], [9E9, 9E9, 9E9, 9E9, 9E9, 9E9]];
	VAR jointtarget CDP_1302 := [[11.62, 36.24, 5.39, 0, 48.37, -34.5], [9E9, 9E9, 9E9, 9E9, 9E9, 9E9]];
	VAR jointtarget CDP_1303 := [[11.64, 36.27, 5.34, 0, 48.39, -34.48], [9E9, 9E9, 9E9, 9E9, 9E9, 9E9]];
	VAR jointtarget CDP_1304 := [[11.66, 36.3, 5.29, 0, 48.41, -34.46], [9E9, 9E9, 9E9, 9E9, 9E9, 9E9]];
	VAR jointtarget CDP_1305 := [[11.68, 36.33, 5.24, 0, 48.43, -34.44], [9E9, 9E9, 9E9, 9E9, 9E9, 9E9]];
	VAR jointtarget CDP_1306 := [[11.7, 36.36, 5.18, 0, 48.45, -34.42], [9E9, 9E9, 9E9, 9E9, 9E9, 9E9]];
	VAR jointtarget CDP_1307 := [[11.72, 36.39, 5.13, 0, 48.48, -34.41], [9E9, 9E9, 9E9, 9E9, 9E9, 9E9]];
	VAR jointtarget CDP_1308 := [[11.74, 36.42, 5.08, 0, 48.5, -34.39], [9E9, 9E9, 9E9, 9E9, 9E9, 9E9]];
	VAR jointtarget CDP_1309 := [[11.76, 36.45, 5.03, 0, 48.52, -34.37], [9E9, 9E9, 9E9, 9E9, 9E9, 9E9]];
	VAR jointtarget CDP_1310 := [[11.77, 36.48, 4.98, 0, 48.54, -34.35], [9E9, 9E9, 9E9, 9E9, 9E9, 9E9]];
	VAR jointtarget CDP_1311 := [[11.79, 36.51, 4.93, 0, 48.56, -34.33], [9E9, 9E9, 9E9, 9E9, 9E9, 9E9]];
	VAR jointtarget CDP_1312 := [[11.81, 36.54, 4.87, 0, 48.58, -34.31], [9E9, 9E9, 9E9, 9E9, 9E9, 9E9]];
	VAR jointtarget CDP_1313 := [[11.83, 36.57, 4.82, 0, 48.61, -34.29], [9E9, 9E9, 9E9, 9E9, 9E9, 9E9]];
	VAR jointtarget CDP_1314 := [[11.85, 36.6, 4.77, 0, 48.63, -34.27], [9E9, 9E9, 9E9, 9E9, 9E9, 9E9]];
	VAR jointtarget CDP_1315 := [[11.87, 36.63, 4.72, 0, 48.65, -34.26], [9E9, 9E9, 9E9, 9E9, 9E9, 9E9]];
	VAR jointtarget CDP_1316 := [[11.89, 36.66, 4.67, 0, 48.67, -34.24], [9E9, 9E9, 9E9, 9E9, 9E9, 9E9]];
	VAR jointtarget CDP_1317 := [[11.91, 36.69, 4.61, 0, 48.69, -34.22], [9E9, 9E9, 9E9, 9E9, 9E9, 9E9]];
	VAR jointtarget CDP_1318 := [[11.92, 36.72, 4.56, 0, 48.72, -34.2], [9E9, 9E9, 9E9, 9E9, 9E9, 9E9]];
	VAR jointtarget CDP_1319 := [[11.94, 36.75, 4.51, 0, 48.74, -34.18], [9E9, 9E9, 9E9, 9E9, 9E9, 9E9]];
	VAR jointtarget CDP_1320 := [[12.05, 36.89, 4.27, 0, 48.84, -40.77], [9E9, 9E9, 9E9, 9E9, 9E9, 9E9]];
	VAR jointtarget CDP_1321 := [[12.18, 37, 4.09, 0, 48.91, -54.03], [9E9, 9E9, 9E9, 9E9, 9E9, 9E9]];
	VAR jointtarget CDP_1322 := [[12.33, 37.06, 3.97, 0, 48.96, -67.26], [9E9, 9E9, 9E9, 9E9, 9E9, 9E9]];
	VAR jointtarget CDP_1323 := [[12.49, 37.09, 3.92, 0, 48.98, -80.49], [9E9, 9E9, 9E9, 9E9, 9E9, 9E9]];
	VAR jointtarget CDP_1324 := [[12.65, 37.08, 3.94, 0, 48.97, -93.72], [9E9, 9E9, 9E9, 9E9, 9E9, 9E9]];
	VAR jointtarget CDP_1325 := [[12.8, 37.03, 4.03, 0, 48.94, -106.95], [9E9, 9E9, 9E9, 9E9, 9E9, 9E9]];
	VAR jointtarget CDP_1326 := [[12.94, 36.94, 4.19, 0, 48.87, -120.2], [9E9, 9E9, 9E9, 9E9, 9E9, 9E9]];
	VAR jointtarget CDP_1327 := [[13.06, 36.82, 4.4, 0, 48.78, -133.47], [9E9, 9E9, 9E9, 9E9, 9E9, 9E9]];
	VAR jointtarget CDP_1328 := [[13.15, 36.67, 4.66, 0, 48.67, -146.77], [9E9, 9E9, 9E9, 9E9, 9E9, 9E9]];
	VAR jointtarget CDP_1329 := [[13.2, 36.5, 4.95, 0, 48.55, -160.1], [9E9, 9E9, 9E9, 9E9, 9E9, 9E9]];
	VAR jointtarget CDP_1330 := [[13.22, 36.32, 5.26, 0, 48.42, -173.47], [9E9, 9E9, 9E9, 9E9, 9E9, 9E9]];
	VAR jointtarget CDP_1331 := [[13.2, 36.14, 5.56, 0, 48.3, -186.88], [9E9, 9E9, 9E9, 9E9, 9E9, 9E9]];
	VAR jointtarget CDP_1332 := [[13.15, 35.98, 5.85, 0, 48.18, -200.32], [9E9, 9E9, 9E9, 9E9, 9E9, 9E9]];
	VAR jointtarget CDP_1333 := [[13.06, 35.83, 6.1, 0, 48.07, -213.8], [9E9, 9E9, 9E9, 9E9, 9E9, 9E9]];
	VAR jointtarget CDP_1334 := [[12.93, 35.71, 6.31, 0, 47.99, -227.31], [9E9, 9E9, 9E9, 9E9, 9E9, 9E9]];
	VAR jointtarget CDP_1335 := [[12.79, 35.62, 6.46, 0, 47.92, -240.84], [9E9, 9E9, 9E9, 9E9, 9E9, 9E9]];
	VAR jointtarget CDP_1336 := [[12.63, 35.57, 6.54, 0, 47.89, -254.39], [9E9, 9E9, 9E9, 9E9, 9E9, 9E9]];
	VAR jointtarget CDP_1337 := [[12.47, 35.57, 6.55, 0, 47.89, -267.94], [9E9, 9E9, 9E9, 9E9, 9E9, 9E9]];
	VAR jointtarget CDP_1338 := [[12.3, 35.6, 6.49, 0, 47.91, -281.49], [9E9, 9E9, 9E9, 9E9, 9E9, 9E9]];
	VAR jointtarget CDP_1339 := [[12.15, 35.68, 6.36, 0, 47.96, -295.03], [9E9, 9E9, 9E9, 9E9, 9E9, 9E9]];
	VAR jointtarget CDP_1340 := [[12.13, 35.69, 6.33, 0, 47.98, -301.75], [9E9, 9E9, 9E9, 9E9, 9E9, 9E9]];
	VAR jointtarget CDP_1341 := [[12.1, 35.71, 6.3, 0, 47.99, -301.78], [9E9, 9E9, 9E9, 9E9, 9E9, 9E9]];
	VAR jointtarget CDP_1342 := [[12.07, 35.73, 6.26, 0, 48, -301.81], [9E9, 9E9, 9E9, 9E9, 9E9, 9E9]];
	VAR jointtarget CDP_1343 := [[12.04, 35.75, 6.23, 0, 48.02, -301.84], [9E9, 9E9, 9E9, 9E9, 9E9, 9E9]];
	VAR jointtarget CDP_1344 := [[12.01, 35.77, 6.2, 0, 48.03, -301.87], [9E9, 9E9, 9E9, 9E9, 9E9, 9E9]];
	VAR jointtarget CDP_1345 := [[11.98, 35.79, 6.16, 0, 48.05, -301.89], [9E9, 9E9, 9E9, 9E9, 9E9, 9E9]];
	VAR jointtarget CDP_1346 := [[11.95, 35.81, 6.13, 0, 48.06, -301.92], [9E9, 9E9, 9E9, 9E9, 9E9, 9E9]];
	VAR jointtarget CDP_1347 := [[11.92, 35.83, 6.1, 0, 48.07, -301.95], [9E9, 9E9, 9E9, 9E9, 9E9, 9E9]];
	VAR jointtarget CDP_1348 := [[11.9, 35.85, 6.07, 0, 48.09, -301.98], [9E9, 9E9, 9E9, 9E9, 9E9, 9E9]];
	VAR jointtarget CDP_1349 := [[11.87, 35.87, 6.03, 0, 48.1, -302.01], [9E9, 9E9, 9E9, 9E9, 9E9, 9E9]];
	VAR jointtarget CDP_1350 := [[11.84, 35.89, 6, 0, 48.11, -302.04], [9E9, 9E9, 9E9, 9E9, 9E9, 9E9]];
	VAR jointtarget CDP_1351 := [[11.81, 35.91, 5.97, 0, 48.13, -302.07], [9E9, 9E9, 9E9, 9E9, 9E9, 9E9]];
	VAR jointtarget CDP_1352 := [[11.78, 35.93, 5.93, 0, 48.14, -302.09], [9E9, 9E9, 9E9, 9E9, 9E9, 9E9]];
	VAR jointtarget CDP_1353 := [[11.75, 35.94, 5.9, 0, 48.16, -302.12], [9E9, 9E9, 9E9, 9E9, 9E9, 9E9]];
	VAR jointtarget CDP_1354 := [[11.73, 35.96, 5.87, 0, 48.17, -302.15], [9E9, 9E9, 9E9, 9E9, 9E9, 9E9]];
	VAR jointtarget CDP_1355 := [[11.7, 35.98, 5.83, 0, 48.18, -302.18], [9E9, 9E9, 9E9, 9E9, 9E9, 9E9]];
	VAR jointtarget CDP_1356 := [[11.67, 36, 5.8, 0, 48.2, -302.21], [9E9, 9E9, 9E9, 9E9, 9E9, 9E9]];
	VAR jointtarget CDP_1357 := [[11.64, 36.02, 5.77, 0, 48.21, -302.24], [9E9, 9E9, 9E9, 9E9, 9E9, 9E9]];
	VAR jointtarget CDP_1358 := [[11.61, 36.04, 5.73, 0, 48.22, -302.27], [9E9, 9E9, 9E9, 9E9, 9E9, 9E9]];
	VAR jointtarget CDP_1359 := [[11.58, 36.06, 5.7, 0, 48.24, -302.29], [9E9, 9E9, 9E9, 9E9, 9E9, 9E9]];
	VAR jointtarget CDP_1360 := [[11.54, 36.09, 5.65, 0, 48.26, -301.24], [9E9, 9E9, 9E9, 9E9, 9E9, 9E9]];
	VAR jointtarget CDP_1361 := [[11.49, 36.12, 5.6, 0, 48.28, -299.1], [9E9, 9E9, 9E9, 9E9, 9E9, 9E9]];
	VAR jointtarget CDP_1362 := [[11.44, 36.15, 5.55, 0, 48.3, -296.95], [9E9, 9E9, 9E9, 9E9, 9E9, 9E9]];
	VAR jointtarget CDP_1363 := [[11.39, 36.17, 5.51, 0, 48.32, -294.81], [9E9, 9E9, 9E9, 9E9, 9E9, 9E9]];
	VAR jointtarget CDP_1364 := [[11.34, 36.2, 5.47, 0, 48.34, -292.67], [9E9, 9E9, 9E9, 9E9, 9E9, 9E9]];
	VAR jointtarget CDP_1365 := [[11.28, 36.22, 5.43, 0, 48.35, -290.53], [9E9, 9E9, 9E9, 9E9, 9E9, 9E9]];
	VAR jointtarget CDP_1366 := [[11.23, 36.24, 5.4, 0, 48.36, -288.38], [9E9, 9E9, 9E9, 9E9, 9E9, 9E9]];
	VAR jointtarget CDP_1367 := [[11.18, 36.25, 5.37, 0, 48.38, -286.24], [9E9, 9E9, 9E9, 9E9, 9E9, 9E9]];
	VAR jointtarget CDP_1368 := [[11.13, 36.27, 5.34, 0, 48.39, -284.1], [9E9, 9E9, 9E9, 9E9, 9E9, 9E9]];
	VAR jointtarget CDP_1369 := [[11.07, 36.28, 5.32, 0, 48.4, -281.96], [9E9, 9E9, 9E9, 9E9, 9E9, 9E9]];
	VAR jointtarget CDP_1370 := [[11.02, 36.29, 5.3, 0, 48.4, -279.82], [9E9, 9E9, 9E9, 9E9, 9E9, 9E9]];
	VAR jointtarget CDP_1371 := [[10.96, 36.3, 5.29, 0, 48.41, -277.69], [9E9, 9E9, 9E9, 9E9, 9E9, 9E9]];
	VAR jointtarget CDP_1372 := [[10.91, 36.31, 5.28, 0, 48.41, -275.55], [9E9, 9E9, 9E9, 9E9, 9E9, 9E9]];
	VAR jointtarget CDP_1373 := [[10.85, 36.31, 5.27, 0, 48.42, -273.41], [9E9, 9E9, 9E9, 9E9, 9E9, 9E9]];
	VAR jointtarget CDP_1374 := [[10.8, 36.31, 5.27, 0, 48.42, -271.27], [9E9, 9E9, 9E9, 9E9, 9E9, 9E9]];
	VAR jointtarget CDP_1375 := [[10.74, 36.31, 5.27, 0, 48.42, -269.13], [9E9, 9E9, 9E9, 9E9, 9E9, 9E9]];
	VAR jointtarget CDP_1376 := [[10.69, 36.31, 5.28, 0, 48.41, -266.99], [9E9, 9E9, 9E9, 9E9, 9E9, 9E9]];
	VAR jointtarget CDP_1377 := [[10.63, 36.3, 5.29, 0, 48.41, -264.85], [9E9, 9E9, 9E9, 9E9, 9E9, 9E9]];
	VAR jointtarget CDP_1378 := [[10.58, 36.29, 5.3, 0, 48.4, -262.71], [9E9, 9E9, 9E9, 9E9, 9E9, 9E9]];
	VAR jointtarget CDP_1379 := [[10.52, 36.28, 5.32, 0, 48.4, -260.58], [9E9, 9E9, 9E9, 9E9, 9E9, 9E9]];
	VAR jointtarget CDP_1380 := [[9.44, 36.08, 5.67, 0, 48.25, -260.56], [9E9, 9E9, 9E9, 9E9, 9E9, 9E9]];
	VAR jointtarget CDP_1381 := [[8.36, 35.89, 5.99, 0, 48.12, -261.64], [9E9, 9E9, 9E9, 9E9, 9E9, 9E9]];
	VAR jointtarget CDP_1382 := [[7.27, 35.73, 6.27, 0, 48, -262.73], [9E9, 9E9, 9E9, 9E9, 9E9, 9E9]];
	VAR jointtarget CDP_1383 := [[6.17, 35.59, 6.5, 0, 47.9, -263.83], [9E9, 9E9, 9E9, 9E9, 9E9, 9E9]];
	VAR jointtarget CDP_1384 := [[5.07, 35.48, 6.7, 0, 47.82, -264.93], [9E9, 9E9, 9E9, 9E9, 9E9, 9E9]];
	VAR jointtarget CDP_1385 := [[3.97, 35.38, 6.86, 0, 47.76, -266.03], [9E9, 9E9, 9E9, 9E9, 9E9, 9E9]];
	VAR jointtarget CDP_1386 := [[2.86, 35.31, 6.98, 0, 47.71, -267.14], [9E9, 9E9, 9E9, 9E9, 9E9, 9E9]];
	VAR jointtarget CDP_1387 := [[1.75, 35.26, 7.06, 0, 47.67, -268.25], [9E9, 9E9, 9E9, 9E9, 9E9, 9E9]];
	VAR jointtarget CDP_1388 := [[0.64, 35.24, 7.11, 0, 47.65, -269.36], [9E9, 9E9, 9E9, 9E9, 9E9, 9E9]];
	VAR jointtarget CDP_1389 := [[-0.47, 35.24, 7.11, 0, 47.65, -270.47], [9E9, 9E9, 9E9, 9E9, 9E9, 9E9]];
	VAR jointtarget CDP_1390 := [[-1.58, 35.26, 7.07, 0, 47.67, -271.58], [9E9, 9E9, 9E9, 9E9, 9E9, 9E9]];
	VAR jointtarget CDP_1391 := [[-2.69, 35.3, 7, 0, 47.7, -272.69], [9E9, 9E9, 9E9, 9E9, 9E9, 9E9]];
	VAR jointtarget CDP_1392 := [[-3.8, 35.37, 6.88, 0, 47.75, -273.8], [9E9, 9E9, 9E9, 9E9, 9E9, 9E9]];
	VAR jointtarget CDP_1393 := [[-4.9, 35.46, 6.73, 0, 47.81, -274.9], [9E9, 9E9, 9E9, 9E9, 9E9, 9E9]];
	VAR jointtarget CDP_1394 := [[-6, 35.57, 6.54, 0, 47.89, -276], [9E9, 9E9, 9E9, 9E9, 9E9, 9E9]];
	VAR jointtarget CDP_1395 := [[-7.1, 35.71, 6.3, 0, 47.99, -277.1], [9E9, 9E9, 9E9, 9E9, 9E9, 9E9]];
	VAR jointtarget CDP_1396 := [[-8.19, 35.87, 6.03, 0, 48.1, -278.19], [9E9, 9E9, 9E9, 9E9, 9E9, 9E9]];
	VAR jointtarget CDP_1397 := [[-9.28, 36.05, 5.72, 0, 48.23, -279.28], [9E9, 9E9, 9E9, 9E9, 9E9, 9E9]];
	VAR jointtarget CDP_1398 := [[-10.36, 36.25, 5.38, 0, 48.37, -280.36], [9E9, 9E9, 9E9, 9E9, 9E9, 9E9]];
	VAR jointtarget CDP_1399 := [[-11.43, 36.48, 4.99, 0, 48.54, -281.43], [9E9, 9E9, 9E9, 9E9, 9E9, 9E9]];
	VAR jointtarget CDP_1400 := [[-11.44, 36.48, 4.98, 0, 48.54, -281.78], [9E9, 9E9, 9E9, 9E9, 9E9, 9E9]];
	VAR jointtarget CDP_1401 := [[-11.46, 36.48, 4.97, 0, 48.54, -282.45], [9E9, 9E9, 9E9, 9E9, 9E9, 9E9]];
	VAR jointtarget CDP_1402 := [[-11.48, 36.49, 4.97, 0, 48.54, -283.13], [9E9, 9E9, 9E9, 9E9, 9E9, 9E9]];
	VAR jointtarget CDP_1403 := [[-11.49, 36.49, 4.96, 0, 48.55, -283.81], [9E9, 9E9, 9E9, 9E9, 9E9, 9E9]];
	VAR jointtarget CDP_1404 := [[-11.51, 36.5, 4.95, 0, 48.55, -284.49], [9E9, 9E9, 9E9, 9E9, 9E9, 9E9]];
	VAR jointtarget CDP_1405 := [[-11.53, 36.5, 4.94, 0, 48.55, -285.17], [9E9, 9E9, 9E9, 9E9, 9E9, 9E9]];
	VAR jointtarget CDP_1406 := [[-11.54, 36.51, 4.94, 0, 48.56, -285.84], [9E9, 9E9, 9E9, 9E9, 9E9, 9E9]];
	VAR jointtarget CDP_1407 := [[-11.56, 36.51, 4.93, 0, 48.56, -286.52], [9E9, 9E9, 9E9, 9E9, 9E9, 9E9]];
	VAR jointtarget CDP_1408 := [[-11.57, 36.52, 4.92, 0, 48.57, -287.2], [9E9, 9E9, 9E9, 9E9, 9E9, 9E9]];
	VAR jointtarget CDP_1409 := [[-11.59, 36.52, 4.91, 0, 48.57, -287.88], [9E9, 9E9, 9E9, 9E9, 9E9, 9E9]];
	VAR jointtarget CDP_1410 := [[-11.6, 36.53, 4.9, 0, 48.57, -288.56], [9E9, 9E9, 9E9, 9E9, 9E9, 9E9]];
	VAR jointtarget CDP_1411 := [[-11.62, 36.53, 4.89, 0, 48.58, -289.23], [9E9, 9E9, 9E9, 9E9, 9E9, 9E9]];
	VAR jointtarget CDP_1412 := [[-11.64, 36.54, 4.88, 0, 48.58, -289.91], [9E9, 9E9, 9E9, 9E9, 9E9, 9E9]];
	VAR jointtarget CDP_1413 := [[-11.65, 36.55, 4.87, 0, 48.59, -290.59], [9E9, 9E9, 9E9, 9E9, 9E9, 9E9]];
	VAR jointtarget CDP_1414 := [[-11.67, 36.55, 4.85, 0, 48.59, -291.27], [9E9, 9E9, 9E9, 9E9, 9E9, 9E9]];
	VAR jointtarget CDP_1415 := [[-11.68, 36.56, 4.84, 0, 48.6, -291.94], [9E9, 9E9, 9E9, 9E9, 9E9, 9E9]];
	VAR jointtarget CDP_1416 := [[-11.7, 36.57, 4.83, 0, 48.6, -292.62], [9E9, 9E9, 9E9, 9E9, 9E9, 9E9]];
	VAR jointtarget CDP_1417 := [[-11.71, 36.57, 4.82, 0, 48.61, -293.3], [9E9, 9E9, 9E9, 9E9, 9E9, 9E9]];
	VAR jointtarget CDP_1418 := [[-11.73, 36.58, 4.81, 0, 48.61, -293.98], [9E9, 9E9, 9E9, 9E9, 9E9, 9E9]];
	VAR jointtarget CDP_1419 := [[-11.74, 36.59, 4.79, 0, 48.62, -294.65], [9E9, 9E9, 9E9, 9E9, 9E9, 9E9]];
	VAR jointtarget CDP_1420 := [[-11.8, 36.62, 4.74, 0, 48.64, -295.04], [9E9, 9E9, 9E9, 9E9, 9E9, 9E9]];
	VAR jointtarget CDP_1421 := [[-11.86, 36.65, 4.68, 0, 48.66, -295.11], [9E9, 9E9, 9E9, 9E9, 9E9, 9E9]];
	VAR jointtarget CDP_1422 := [[-11.93, 36.68, 4.63, 0, 48.69, -295.17], [9E9, 9E9, 9E9, 9E9, 9E9, 9E9]];
	VAR jointtarget CDP_1423 := [[-11.99, 36.71, 4.58, 0, 48.71, -295.23], [9E9, 9E9, 9E9, 9E9, 9E9, 9E9]];
	VAR jointtarget CDP_1424 := [[-12.05, 36.75, 4.52, 0, 48.73, -295.29], [9E9, 9E9, 9E9, 9E9, 9E9, 9E9]];
	VAR jointtarget CDP_1425 := [[-12.11, 36.78, 4.47, 0, 48.75, -295.35], [9E9, 9E9, 9E9, 9E9, 9E9, 9E9]];
	VAR jointtarget CDP_1426 := [[-12.17, 36.81, 4.41, 0, 48.78, -295.41], [9E9, 9E9, 9E9, 9E9, 9E9, 9E9]];
	VAR jointtarget CDP_1427 := [[-12.23, 36.84, 4.36, 0, 48.8, -295.47], [9E9, 9E9, 9E9, 9E9, 9E9, 9E9]];
	VAR jointtarget CDP_1428 := [[-12.29, 36.87, 4.3, 0, 48.82, -295.53], [9E9, 9E9, 9E9, 9E9, 9E9, 9E9]];
	VAR jointtarget CDP_1429 := [[-12.35, 36.9, 4.25, 0, 48.85, -295.59], [9E9, 9E9, 9E9, 9E9, 9E9, 9E9]];
	VAR jointtarget CDP_1430 := [[-12.41, 36.94, 4.19, 0, 48.87, -295.65], [9E9, 9E9, 9E9, 9E9, 9E9, 9E9]];
	VAR jointtarget CDP_1431 := [[-12.47, 36.97, 4.14, 0, 48.89, -295.71], [9E9, 9E9, 9E9, 9E9, 9E9, 9E9]];
	VAR jointtarget CDP_1432 := [[-12.53, 37, 4.08, 0, 48.92, -295.77], [9E9, 9E9, 9E9, 9E9, 9E9, 9E9]];
	VAR jointtarget CDP_1433 := [[-12.59, 37.03, 4.03, 0, 48.94, -295.83], [9E9, 9E9, 9E9, 9E9, 9E9, 9E9]];
	VAR jointtarget CDP_1434 := [[-12.65, 37.07, 3.97, 0, 48.96, -295.89], [9E9, 9E9, 9E9, 9E9, 9E9, 9E9]];
	VAR jointtarget CDP_1435 := [[-12.71, 37.1, 3.92, 0, 48.99, -295.95], [9E9, 9E9, 9E9, 9E9, 9E9, 9E9]];
	VAR jointtarget CDP_1436 := [[-12.77, 37.13, 3.86, 0, 49.01, -296.01], [9E9, 9E9, 9E9, 9E9, 9E9, 9E9]];
	VAR jointtarget CDP_1437 := [[-12.83, 37.16, 3.8, 0, 49.03, -296.07], [9E9, 9E9, 9E9, 9E9, 9E9, 9E9]];
	VAR jointtarget CDP_1438 := [[-12.89, 37.2, 3.75, 0, 49.06, -296.13], [9E9, 9E9, 9E9, 9E9, 9E9, 9E9]];
	VAR jointtarget CDP_1439 := [[-12.95, 37.23, 3.69, 0, 49.08, -296.19], [9E9, 9E9, 9E9, 9E9, 9E9, 9E9]];
	VAR jointtarget CDP_1440 := [[-13.07, 37.28, 3.6, 0, 49.12, -291.14], [9E9, 9E9, 9E9, 9E9, 9E9, 9E9]];
	VAR jointtarget CDP_1441 := [[-13.19, 37.31, 3.56, 0, 49.14, -280.95], [9E9, 9E9, 9E9, 9E9, 9E9, 9E9]];
	VAR jointtarget CDP_1442 := [[-13.32, 37.31, 3.55, 0, 49.14, -270.75], [9E9, 9E9, 9E9, 9E9, 9E9, 9E9]];
	VAR jointtarget CDP_1443 := [[-13.45, 37.28, 3.59, 0, 49.12, -260.55], [9E9, 9E9, 9E9, 9E9, 9E9, 9E9]];
	VAR jointtarget CDP_1444 := [[-13.57, 37.24, 3.68, 0, 49.09, -250.35], [9E9, 9E9, 9E9, 9E9, 9E9, 9E9]];
	VAR jointtarget CDP_1445 := [[-13.68, 37.16, 3.8, 0, 49.03, -240.14], [9E9, 9E9, 9E9, 9E9, 9E9, 9E9]];
	VAR jointtarget CDP_1446 := [[-13.78, 37.07, 3.96, 0, 48.97, -229.91], [9E9, 9E9, 9E9, 9E9, 9E9, 9E9]];
	VAR jointtarget CDP_1447 := [[-13.86, 36.96, 4.15, 0, 48.89, -219.67], [9E9, 9E9, 9E9, 9E9, 9E9, 9E9]];
	VAR jointtarget CDP_1448 := [[-13.93, 36.84, 4.37, 0, 48.8, -209.41], [9E9, 9E9, 9E9, 9E9, 9E9, 9E9]];
	VAR jointtarget CDP_1449 := [[-13.97, 36.7, 4.6, 0, 48.7, -199.13], [9E9, 9E9, 9E9, 9E9, 9E9, 9E9]];
	VAR jointtarget CDP_1450 := [[-13.99, 36.56, 4.85, 0, 48.6, -188.83], [9E9, 9E9, 9E9, 9E9, 9E9, 9E9]];
	VAR jointtarget CDP_1451 := [[-13.98, 36.42, 5.09, 0, 48.49, -178.5], [9E9, 9E9, 9E9, 9E9, 9E9, 9E9]];
	VAR jointtarget CDP_1452 := [[-13.96, 36.28, 5.33, 0, 48.39, -168.15], [9E9, 9E9, 9E9, 9E9, 9E9, 9E9]];
	VAR jointtarget CDP_1453 := [[-13.91, 36.14, 5.56, 0, 48.3, -157.77], [9E9, 9E9, 9E9, 9E9, 9E9, 9E9]];
	VAR jointtarget CDP_1454 := [[-13.84, 36.02, 5.77, 0, 48.21, -147.38], [9E9, 9E9, 9E9, 9E9, 9E9, 9E9]];
	VAR jointtarget CDP_1455 := [[-13.75, 35.92, 5.94, 0, 48.14, -136.97], [9E9, 9E9, 9E9, 9E9, 9E9, 9E9]];
	VAR jointtarget CDP_1456 := [[-13.64, 35.83, 6.09, 0, 48.08, -126.54], [9E9, 9E9, 9E9, 9E9, 9E9, 9E9]];
	VAR jointtarget CDP_1457 := [[-13.52, 35.77, 6.2, 0, 48.03, -116.09], [9E9, 9E9, 9E9, 9E9, 9E9, 9E9]];
	VAR jointtarget CDP_1458 := [[-13.4, 35.73, 6.26, 0, 48, -105.64], [9E9, 9E9, 9E9, 9E9, 9E9, 9E9]];
	VAR jointtarget CDP_1459 := [[-13.27, 35.72, 6.28, 0, 48, -95.19], [9E9, 9E9, 9E9, 9E9, 9E9, 9E9]];
	VAR jointtarget CDP_1460 := [[-13.2, 35.72, 6.28, 0, 48, -89.96], [9E9, 9E9, 9E9, 9E9, 9E9, 9E9]];
	VAR jointtarget CDP_1461 := [[-13.13, 35.72, 6.28, 0, 48, -89.89], [9E9, 9E9, 9E9, 9E9, 9E9, 9E9]];
	VAR jointtarget CDP_1462 := [[-13.06, 35.72, 6.28, 0, 48, -89.82], [9E9, 9E9, 9E9, 9E9, 9E9, 9E9]];
	VAR jointtarget CDP_1463 := [[-12.99, 35.72, 6.28, 0, 48, -89.75], [9E9, 9E9, 9E9, 9E9, 9E9, 9E9]];
	VAR jointtarget CDP_1464 := [[-12.93, 35.72, 6.28, 0, 48, -89.69], [9E9, 9E9, 9E9, 9E9, 9E9, 9E9]];
	VAR jointtarget CDP_1465 := [[-12.86, 35.72, 6.28, 0, 48, -89.62], [9E9, 9E9, 9E9, 9E9, 9E9, 9E9]];
	VAR jointtarget CDP_1466 := [[-12.79, 35.72, 6.28, 0, 48, -89.55], [9E9, 9E9, 9E9, 9E9, 9E9, 9E9]];
	VAR jointtarget CDP_1467 := [[-12.72, 35.72, 6.28, 0, 48, -89.48], [9E9, 9E9, 9E9, 9E9, 9E9, 9E9]];
	VAR jointtarget CDP_1468 := [[-12.65, 35.72, 6.28, 0, 48, -89.41], [9E9, 9E9, 9E9, 9E9, 9E9, 9E9]];
	VAR jointtarget CDP_1469 := [[-12.59, 35.72, 6.28, 0, 48, -89.35], [9E9, 9E9, 9E9, 9E9, 9E9, 9E9]];
	VAR jointtarget CDP_1470 := [[-12.52, 35.72, 6.28, 0, 48.01, -89.28], [9E9, 9E9, 9E9, 9E9, 9E9, 9E9]];
	VAR jointtarget CDP_1471 := [[-12.45, 35.72, 6.27, 0, 48.01, -89.21], [9E9, 9E9, 9E9, 9E9, 9E9, 9E9]];
	VAR jointtarget CDP_1472 := [[-12.38, 35.72, 6.27, 0, 48.01, -89.14], [9E9, 9E9, 9E9, 9E9, 9E9, 9E9]];
	VAR jointtarget CDP_1473 := [[-12.32, 35.72, 6.27, 0, 48.01, -89.07], [9E9, 9E9, 9E9, 9E9, 9E9, 9E9]];
	VAR jointtarget CDP_1474 := [[-12.25, 35.72, 6.27, 0, 48.01, -89.01], [9E9, 9E9, 9E9, 9E9, 9E9, 9E9]];
	VAR jointtarget CDP_1475 := [[-12.18, 35.72, 6.27, 0, 48.01, -88.94], [9E9, 9E9, 9E9, 9E9, 9E9, 9E9]];
	VAR jointtarget CDP_1476 := [[-12.11, 35.72, 6.26, 0, 48.02, -88.87], [9E9, 9E9, 9E9, 9E9, 9E9, 9E9]];
	VAR jointtarget CDP_1477 := [[-12.04, 35.72, 6.26, 0, 48.02, -88.8], [9E9, 9E9, 9E9, 9E9, 9E9, 9E9]];
	VAR jointtarget CDP_1478 := [[-11.98, 35.72, 6.26, 0, 48.02, -88.74], [9E9, 9E9, 9E9, 9E9, 9E9, 9E9]];
	VAR jointtarget CDP_1479 := [[-11.91, 35.72, 6.25, 0, 48.02, -88.67], [9E9, 9E9, 9E9, 9E9, 9E9, 9E9]];
	VAR jointtarget CDP_1480 := [[-11.89, 35.72, 6.25, 0, 48.02, -88.98], [9E9, 9E9, 9E9, 9E9, 9E9, 9E9]];
	VAR jointtarget CDP_1481 := [[-11.87, 35.72, 6.25, 0, 48.02, -89.63], [9E9, 9E9, 9E9, 9E9, 9E9, 9E9]];
	VAR jointtarget CDP_1482 := [[-11.86, 35.72, 6.25, 0, 48.02, -90.27], [9E9, 9E9, 9E9, 9E9, 9E9, 9E9]];
	VAR jointtarget CDP_1483 := [[-11.84, 35.72, 6.25, 0, 48.02, -90.92], [9E9, 9E9, 9E9, 9E9, 9E9, 9E9]];
	VAR jointtarget CDP_1484 := [[-11.82, 35.72, 6.25, 0, 48.02, -91.56], [9E9, 9E9, 9E9, 9E9, 9E9, 9E9]];
	VAR jointtarget CDP_1485 := [[-11.81, 35.72, 6.26, 0, 48.02, -92.21], [9E9, 9E9, 9E9, 9E9, 9E9, 9E9]];
	VAR jointtarget CDP_1486 := [[-11.79, 35.72, 6.26, 0, 48.02, -92.85], [9E9, 9E9, 9E9, 9E9, 9E9, 9E9]];
	VAR jointtarget CDP_1487 := [[-11.77, 35.72, 6.26, 0, 48.02, -93.5], [9E9, 9E9, 9E9, 9E9, 9E9, 9E9]];
	VAR jointtarget CDP_1488 := [[-11.76, 35.72, 6.26, 0, 48.02, -94.14], [9E9, 9E9, 9E9, 9E9, 9E9, 9E9]];
	VAR jointtarget CDP_1489 := [[-11.74, 35.72, 6.26, 0, 48.02, -94.79], [9E9, 9E9, 9E9, 9E9, 9E9, 9E9]];
	VAR jointtarget CDP_1490 := [[-11.72, 35.72, 6.27, 0, 48.02, -95.43], [9E9, 9E9, 9E9, 9E9, 9E9, 9E9]];
	VAR jointtarget CDP_1491 := [[-11.71, 35.71, 6.27, 0, 48.02, -96.08], [9E9, 9E9, 9E9, 9E9, 9E9, 9E9]];
	VAR jointtarget CDP_1492 := [[-11.69, 35.71, 6.27, 0, 48.01, -96.72], [9E9, 9E9, 9E9, 9E9, 9E9, 9E9]];
	VAR jointtarget CDP_1493 := [[-11.67, 35.71, 6.28, 0, 48.01, -97.37], [9E9, 9E9, 9E9, 9E9, 9E9, 9E9]];
	VAR jointtarget CDP_1494 := [[-11.66, 35.71, 6.28, 0, 48.01, -98.01], [9E9, 9E9, 9E9, 9E9, 9E9, 9E9]];
	VAR jointtarget CDP_1495 := [[-11.64, 35.7, 6.29, 0, 48.01, -98.66], [9E9, 9E9, 9E9, 9E9, 9E9, 9E9]];
	VAR jointtarget CDP_1496 := [[-11.62, 35.7, 6.29, 0, 48.01, -99.31], [9E9, 9E9, 9E9, 9E9, 9E9, 9E9]];
	VAR jointtarget CDP_1497 := [[-11.61, 35.7, 6.3, 0, 48, -99.95], [9E9, 9E9, 9E9, 9E9, 9E9, 9E9]];
	VAR jointtarget CDP_1498 := [[-11.59, 35.69, 6.3, 0, 48, -100.6], [9E9, 9E9, 9E9, 9E9, 9E9, 9E9]];
	VAR jointtarget CDP_1499 := [[-11.57, 35.69, 6.31, 0, 48, -101.24], [9E9, 9E9, 9E9, 9E9, 9E9, 9E9]];
	VAR jointtarget CDP_1500 := [[-10.48, 35.46, 6.7, 0, 47.84, -100.48], [9E9, 9E9, 9E9, 9E9, 9E9, 9E9]];
	VAR jointtarget CDP_1501 := [[-9.38, 35.26, 7.05, 0, 47.69, -99.38], [9E9, 9E9, 9E9, 9E9, 9E9, 9E9]];
	VAR jointtarget CDP_1502 := [[-8.27, 35.07, 7.37, 0, 47.56, -98.27], [9E9, 9E9, 9E9, 9E9, 9E9, 9E9]];
	VAR jointtarget CDP_1503 := [[-7.15, 34.91, 7.64, 0, 47.45, -97.15], [9E9, 9E9, 9E9, 9E9, 9E9, 9E9]];
	VAR jointtarget CDP_1504 := [[-6.03, 34.78, 7.87, 0, 47.35, -96.03], [9E9, 9E9, 9E9, 9E9, 9E9, 9E9]];
	VAR jointtarget CDP_1505 := [[-4.9, 34.66, 8.06, 0, 47.27, -94.9], [9E9, 9E9, 9E9, 9E9, 9E9, 9E9]];
	VAR jointtarget CDP_1506 := [[-3.77, 34.57, 8.22, 0, 47.21, -93.77], [9E9, 9E9, 9E9, 9E9, 9E9, 9E9]];
	VAR jointtarget CDP_1507 := [[-2.64, 34.51, 8.33, 0, 47.16, -92.64], [9E9, 9E9, 9E9, 9E9, 9E9, 9E9]];
	VAR jointtarget CDP_1508 := [[-1.51, 34.46, 8.4, 0, 47.13, -91.51], [9E9, 9E9, 9E9, 9E9, 9E9, 9E9]];
	VAR jointtarget CDP_1509 := [[-0.37, 34.44, 8.44, 0, 47.12, -90.37], [9E9, 9E9, 9E9, 9E9, 9E9, 9E9]];
	VAR jointtarget CDP_1510 := [[0.76, 34.45, 8.43, 0, 47.12, -89.24], [9E9, 9E9, 9E9, 9E9, 9E9, 9E9]];
	VAR jointtarget CDP_1511 := [[1.9, 34.48, 8.38, 0, 47.14, -88.1], [9E9, 9E9, 9E9, 9E9, 9E9, 9E9]];
	VAR jointtarget CDP_1512 := [[3.03, 34.53, 8.3, 0, 47.18, -86.97], [9E9, 9E9, 9E9, 9E9, 9E9, 9E9]];
	VAR jointtarget CDP_1513 := [[4.16, 34.6, 8.17, 0, 47.23, -85.84], [9E9, 9E9, 9E9, 9E9, 9E9, 9E9]];
	VAR jointtarget CDP_1514 := [[5.29, 34.7, 8, 0, 47.3, -84.71], [9E9, 9E9, 9E9, 9E9, 9E9, 9E9]];
	VAR jointtarget CDP_1515 := [[6.42, 34.82, 7.79, 0, 47.38, -83.58], [9E9, 9E9, 9E9, 9E9, 9E9, 9E9]];
	VAR jointtarget CDP_1516 := [[7.54, 34.97, 7.55, 0, 47.49, -82.46], [9E9, 9E9, 9E9, 9E9, 9E9, 9E9]];
	VAR jointtarget CDP_1517 := [[8.65, 35.13, 7.26, 0, 47.6, -81.35], [9E9, 9E9, 9E9, 9E9, 9E9, 9E9]];
	VAR jointtarget CDP_1518 := [[9.76, 35.32, 6.94, 0, 47.74, -80.24], [9E9, 9E9, 9E9, 9E9, 9E9, 9E9]];
	VAR jointtarget CDP_1519 := [[10.86, 35.54, 6.57, 0, 47.89, -79.14], [9E9, 9E9, 9E9, 9E9, 9E9, 9E9]];
	VAR jointtarget CDP_1520 := [[10.87, 35.54, 6.56, 0, 47.89, -79.46], [9E9, 9E9, 9E9, 9E9, 9E9, 9E9]];
	VAR jointtarget CDP_1521 := [[10.89, 35.54, 6.56, 0, 47.9, -80.1], [9E9, 9E9, 9E9, 9E9, 9E9, 9E9]];
	VAR jointtarget CDP_1522 := [[10.91, 35.55, 6.55, 0, 47.9, -80.75], [9E9, 9E9, 9E9, 9E9, 9E9, 9E9]];
	VAR jointtarget CDP_1523 := [[10.92, 35.55, 6.55, 0, 47.9, -81.39], [9E9, 9E9, 9E9, 9E9, 9E9, 9E9]];
	VAR jointtarget CDP_1524 := [[10.94, 35.55, 6.55, 0, 47.9, -82.04], [9E9, 9E9, 9E9, 9E9, 9E9, 9E9]];
	VAR jointtarget CDP_1525 := [[10.96, 35.56, 6.54, 0, 47.9, -82.68], [9E9, 9E9, 9E9, 9E9, 9E9, 9E9]];
	VAR jointtarget CDP_1526 := [[10.97, 35.56, 6.54, 0, 47.9, -83.33], [9E9, 9E9, 9E9, 9E9, 9E9, 9E9]];
	VAR jointtarget CDP_1527 := [[10.99, 35.56, 6.53, 0, 47.91, -83.97], [9E9, 9E9, 9E9, 9E9, 9E9, 9E9]];
	VAR jointtarget CDP_1528 := [[11.01, 35.56, 6.53, 0, 47.91, -84.62], [9E9, 9E9, 9E9, 9E9, 9E9, 9E9]];
	VAR jointtarget CDP_1529 := [[11.02, 35.56, 6.53, 0, 47.91, -85.27], [9E9, 9E9, 9E9, 9E9, 9E9, 9E9]];
	VAR jointtarget CDP_1530 := [[11.04, 35.56, 6.53, 0, 47.91, -85.91], [9E9, 9E9, 9E9, 9E9, 9E9, 9E9]];
	VAR jointtarget CDP_1531 := [[11.06, 35.56, 6.53, 0, 47.91, -86.56], [9E9, 9E9, 9E9, 9E9, 9E9, 9E9]];
	VAR jointtarget CDP_1532 := [[11.07, 35.57, 6.52, 0, 47.91, -87.2], [9E9, 9E9, 9E9, 9E9, 9E9, 9E9]];
	VAR jointtarget CDP_1533 := [[11.09, 35.57, 6.52, 0, 47.91, -87.85], [9E9, 9E9, 9E9, 9E9, 9E9, 9E9]];
	VAR jointtarget CDP_1534 := [[11.11, 35.57, 6.52, 0, 47.91, -88.49], [9E9, 9E9, 9E9, 9E9, 9E9, 9E9]];
	VAR jointtarget CDP_1535 := [[11.13, 35.57, 6.52, 0, 47.91, -89.14], [9E9, 9E9, 9E9, 9E9, 9E9, 9E9]];
	VAR jointtarget CDP_1536 := [[11.14, 35.57, 6.52, 0, 47.91, -89.78], [9E9, 9E9, 9E9, 9E9, 9E9, 9E9]];
	VAR jointtarget CDP_1537 := [[11.16, 35.57, 6.52, 0, 47.91, -90.43], [9E9, 9E9, 9E9, 9E9, 9E9, 9E9]];
	VAR jointtarget CDP_1538 := [[11.18, 35.57, 6.52, 0, 47.91, -91.07], [9E9, 9E9, 9E9, 9E9, 9E9, 9E9]];
	VAR jointtarget CDP_1539 := [[11.19, 35.57, 6.52, 0, 47.91, -91.72], [9E9, 9E9, 9E9, 9E9, 9E9, 9E9]];
	VAR jointtarget CDP_1540 := [[11.26, 35.56, 6.53, 0, 47.91, -91.98], [9E9, 9E9, 9E9, 9E9, 9E9, 9E9]];
	VAR jointtarget CDP_1541 := [[11.33, 35.56, 6.53, 0, 47.91, -91.91], [9E9, 9E9, 9E9, 9E9, 9E9, 9E9]];
	VAR jointtarget CDP_1542 := [[11.4, 35.56, 6.54, 0, 47.91, -91.84], [9E9, 9E9, 9E9, 9E9, 9E9, 9E9]];
	VAR jointtarget CDP_1543 := [[11.47, 35.56, 6.54, 0, 47.9, -91.78], [9E9, 9E9, 9E9, 9E9, 9E9, 9E9]];
	VAR jointtarget CDP_1544 := [[11.53, 35.55, 6.54, 0, 47.9, -91.71], [9E9, 9E9, 9E9, 9E9, 9E9, 9E9]];
	VAR jointtarget CDP_1545 := [[11.6, 35.55, 6.55, 0, 47.9, -91.64], [9E9, 9E9, 9E9, 9E9, 9E9, 9E9]];
	VAR jointtarget CDP_1546 := [[11.67, 35.55, 6.55, 0, 47.9, -91.57], [9E9, 9E9, 9E9, 9E9, 9E9, 9E9]];
	VAR jointtarget CDP_1547 := [[11.74, 35.55, 6.55, 0, 47.9, -91.5], [9E9, 9E9, 9E9, 9E9, 9E9, 9E9]];
	VAR jointtarget CDP_1548 := [[11.81, 35.55, 6.56, 0, 47.9, -91.44], [9E9, 9E9, 9E9, 9E9, 9E9, 9E9]];
	VAR jointtarget CDP_1549 := [[11.87, 35.54, 6.56, 0, 47.9, -91.37], [9E9, 9E9, 9E9, 9E9, 9E9, 9E9]];
	VAR jointtarget CDP_1550 := [[11.94, 35.54, 6.56, 0, 47.89, -91.3], [9E9, 9E9, 9E9, 9E9, 9E9, 9E9]];
	VAR jointtarget CDP_1551 := [[12.01, 35.54, 6.57, 0, 47.89, -91.23], [9E9, 9E9, 9E9, 9E9, 9E9, 9E9]];
	VAR jointtarget CDP_1552 := [[12.08, 35.54, 6.57, 0, 47.89, -91.16], [9E9, 9E9, 9E9, 9E9, 9E9, 9E9]];
	VAR jointtarget CDP_1553 := [[12.15, 35.54, 6.57, 0, 47.89, -91.09], [9E9, 9E9, 9E9, 9E9, 9E9, 9E9]];
	VAR jointtarget CDP_1554 := [[12.21, 35.54, 6.57, 0, 47.89, -91.03], [9E9, 9E9, 9E9, 9E9, 9E9, 9E9]];
	VAR jointtarget CDP_1555 := [[12.28, 35.54, 6.58, 0, 47.89, -90.96], [9E9, 9E9, 9E9, 9E9, 9E9, 9E9]];
	VAR jointtarget CDP_1556 := [[12.35, 35.53, 6.58, 0, 47.89, -90.89], [9E9, 9E9, 9E9, 9E9, 9E9, 9E9]];
	VAR jointtarget CDP_1557 := [[12.42, 35.53, 6.58, 0, 47.89, -90.82], [9E9, 9E9, 9E9, 9E9, 9E9, 9E9]];
	VAR jointtarget CDP_1558 := [[12.49, 35.53, 6.58, 0, 47.89, -90.75], [9E9, 9E9, 9E9, 9E9, 9E9, 9E9]];
	VAR jointtarget CDP_1559 := [[12.55, 35.53, 6.58, 0, 47.89, -90.69], [9E9, 9E9, 9E9, 9E9, 9E9, 9E9]];
	VAR jointtarget CDP_1560 := [[12.69, 35.54, 6.56, 0, 47.89, -85.39], [9E9, 9E9, 9E9, 9E9, 9E9, 9E9]];
	VAR jointtarget CDP_1561 := [[12.81, 35.58, 6.5, 0, 47.92, -74.94], [9E9, 9E9, 9E9, 9E9, 9E9, 9E9]];
	VAR jointtarget CDP_1562 := [[12.93, 35.64, 6.4, 0, 47.96, -64.5], [9E9, 9E9, 9E9, 9E9, 9E9, 9E9]];
	VAR jointtarget CDP_1563 := [[13.04, 35.72, 6.25, 0, 48.02, -54.07], [9E9, 9E9, 9E9, 9E9, 9E9, 9E9]];
	VAR jointtarget CDP_1564 := [[13.13, 35.83, 6.08, 0, 48.1, -43.65], [9E9, 9E9, 9E9, 9E9, 9E9, 9E9]];
	VAR jointtarget CDP_1565 := [[13.2, 35.95, 5.87, 0, 48.18, -33.25], [9E9, 9E9, 9E9, 9E9, 9E9, 9E9]];
	VAR jointtarget CDP_1566 := [[13.25, 36.08, 5.65, 0, 48.28, -22.88], [9E9, 9E9, 9E9, 9E9, 9E9, 9E9]];
	VAR jointtarget CDP_1567 := [[13.28, 36.22, 5.41, 0, 48.37, -12.53], [9E9, 9E9, 9E9, 9E9, 9E9, 9E9]];
	VAR jointtarget CDP_1568 := [[13.29, 36.36, 5.16, 0, 48.48, -2.2], [9E9, 9E9, 9E9, 9E9, 9E9, 9E9]];
	VAR jointtarget CDP_1569 := [[13.27, 36.5, 4.92, 0, 48.58, 8.11], [9E9, 9E9, 9E9, 9E9, 9E9, 9E9]];
	VAR jointtarget CDP_1570 := [[13.23, 36.64, 4.69, 0, 48.68, 18.39], [9E9, 9E9, 9E9, 9E9, 9E9, 9E9]];
	VAR jointtarget CDP_1571 := [[13.17, 36.76, 4.47, 0, 48.77, 28.65], [9E9, 9E9, 9E9, 9E9, 9E9, 9E9]];
	VAR jointtarget CDP_1572 := [[13.08, 36.87, 4.28, 0, 48.85, 38.9], [9E9, 9E9, 9E9, 9E9, 9E9, 9E9]];
	VAR jointtarget CDP_1573 := [[12.99, 36.97, 4.12, 0, 48.92, 49.12], [9E9, 9E9, 9E9, 9E9, 9E9, 9E9]];
	VAR jointtarget CDP_1574 := [[12.88, 37.04, 3.99, 0, 48.97, 59.33], [9E9, 9E9, 9E9, 9E9, 9E9, 9E9]];
	VAR jointtarget CDP_1575 := [[12.75, 37.09, 3.9, 0, 49.01, 69.54], [9E9, 9E9, 9E9, 9E9, 9E9, 9E9]];
	VAR jointtarget CDP_1576 := [[12.63, 37.12, 3.86, 0, 49.02, 79.73], [9E9, 9E9, 9E9, 9E9, 9E9, 9E9]];
	VAR jointtarget CDP_1577 := [[12.5, 37.12, 3.86, 0, 49.02, 89.93], [9E9, 9E9, 9E9, 9E9, 9E9, 9E9]];
	VAR jointtarget CDP_1578 := [[12.37, 37.09, 3.9, 0, 49.01, 100.13], [9E9, 9E9, 9E9, 9E9, 9E9, 9E9]];
	VAR jointtarget CDP_1579 := [[12.25, 37.04, 3.99, 0, 48.97, 110.33], [9E9, 9E9, 9E9, 9E9, 9E9, 9E9]];
	VAR jointtarget CDP_1580 := [[12.19, 37.01, 4.04, 0, 48.95, 115.43], [9E9, 9E9, 9E9, 9E9, 9E9, 9E9]];
	VAR jointtarget CDP_1581 := [[12.13, 36.98, 4.1, 0, 48.92, 115.37], [9E9, 9E9, 9E9, 9E9, 9E9, 9E9]];
	VAR jointtarget CDP_1582 := [[12.07, 36.95, 4.15, 0, 48.9, 115.31], [9E9, 9E9, 9E9, 9E9, 9E9, 9E9]];
	VAR jointtarget CDP_1583 := [[12.01, 36.91, 4.21, 0, 48.88, 115.25], [9E9, 9E9, 9E9, 9E9, 9E9, 9E9]];
	VAR jointtarget CDP_1584 := [[11.95, 36.88, 4.26, 0, 48.85, 115.19], [9E9, 9E9, 9E9, 9E9, 9E9, 9E9]];
	VAR jointtarget CDP_1585 := [[11.89, 36.85, 4.32, 0, 48.83, 115.13], [9E9, 9E9, 9E9, 9E9, 9E9, 9E9]];
	VAR jointtarget CDP_1586 := [[11.83, 36.82, 4.37, 0, 48.81, 115.07], [9E9, 9E9, 9E9, 9E9, 9E9, 9E9]];
	VAR jointtarget CDP_1587 := [[11.77, 36.79, 4.42, 0, 48.79, 115.01], [9E9, 9E9, 9E9, 9E9, 9E9, 9E9]];
	VAR jointtarget CDP_1588 := [[11.71, 36.76, 4.48, 0, 48.76, 114.95], [9E9, 9E9, 9E9, 9E9, 9E9, 9E9]];
	VAR jointtarget CDP_1589 := [[11.65, 36.73, 4.53, 0, 48.74, 114.89], [9E9, 9E9, 9E9, 9E9, 9E9, 9E9]];
	VAR jointtarget CDP_1590 := [[11.59, 36.7, 4.58, 0, 48.72, 114.83], [9E9, 9E9, 9E9, 9E9, 9E9, 9E9]];
	VAR jointtarget CDP_1591 := [[11.53, 36.67, 4.64, 0, 48.7, 114.77], [9E9, 9E9, 9E9, 9E9, 9E9, 9E9]];
	VAR jointtarget CDP_1592 := [[11.47, 36.63, 4.69, 0, 48.68, 114.71], [9E9, 9E9, 9E9, 9E9, 9E9, 9E9]];
	VAR jointtarget CDP_1593 := [[11.4, 36.6, 4.74, 0, 48.65, 114.64], [9E9, 9E9, 9E9, 9E9, 9E9, 9E9]];
	VAR jointtarget CDP_1594 := [[11.34, 36.57, 4.8, 0, 48.63, 114.58], [9E9, 9E9, 9E9, 9E9, 9E9, 9E9]];
	VAR jointtarget CDP_1595 := [[11.28, 36.54, 4.85, 0, 48.61, 114.52], [9E9, 9E9, 9E9, 9E9, 9E9, 9E9]];
	VAR jointtarget CDP_1596 := [[11.22, 36.51, 4.9, 0, 48.59, 114.46], [9E9, 9E9, 9E9, 9E9, 9E9, 9E9]];
	VAR jointtarget CDP_1597 := [[11.16, 36.48, 4.95, 0, 48.56, 114.4], [9E9, 9E9, 9E9, 9E9, 9E9, 9E9]];
	VAR jointtarget CDP_1598 := [[11.1, 36.45, 5.01, 0, 48.54, 114.34], [9E9, 9E9, 9E9, 9E9, 9E9, 9E9]];
	VAR jointtarget CDP_1599 := [[11.04, 36.42, 5.06, 0, 48.52, 114.28], [9E9, 9E9, 9E9, 9E9, 9E9, 9E9]];
	VAR jointtarget CDP_1600 := [[11.02, 36.41, 5.07, 0, 48.52, 113.93], [9E9, 9E9, 9E9, 9E9, 9E9, 9E9]];
	VAR jointtarget CDP_1601 := [[11.01, 36.41, 5.08, 0, 48.51, 113.26], [9E9, 9E9, 9E9, 9E9, 9E9, 9E9]];
	VAR jointtarget CDP_1602 := [[10.99, 36.4, 5.1, 0, 48.51, 112.58], [9E9, 9E9, 9E9, 9E9, 9E9, 9E9]];
	VAR jointtarget CDP_1603 := [[10.98, 36.39, 5.11, 0, 48.5, 111.9], [9E9, 9E9, 9E9, 9E9, 9E9, 9E9]];
	VAR jointtarget CDP_1604 := [[10.96, 36.39, 5.12, 0, 48.5, 111.22], [9E9, 9E9, 9E9, 9E9, 9E9, 9E9]];
	VAR jointtarget CDP_1605 := [[10.95, 36.38, 5.13, 0, 48.49, 110.55], [9E9, 9E9, 9E9, 9E9, 9E9, 9E9]];
	VAR jointtarget CDP_1606 := [[10.93, 36.37, 5.14, 0, 48.49, 109.87], [9E9, 9E9, 9E9, 9E9, 9E9, 9E9]];
	VAR jointtarget CDP_1607 := [[10.91, 36.37, 5.15, 0, 48.48, 109.19], [9E9, 9E9, 9E9, 9E9, 9E9, 9E9]];
	VAR jointtarget CDP_1608 := [[10.9, 36.36, 5.16, 0, 48.48, 108.51], [9E9, 9E9, 9E9, 9E9, 9E9, 9E9]];
	VAR jointtarget CDP_1609 := [[10.88, 36.36, 5.17, 0, 48.47, 107.83], [9E9, 9E9, 9E9, 9E9, 9E9, 9E9]];
	VAR jointtarget CDP_1610 := [[10.87, 36.35, 5.18, 0, 48.47, 107.16], [9E9, 9E9, 9E9, 9E9, 9E9, 9E9]];
	VAR jointtarget CDP_1611 := [[10.85, 36.34, 5.19, 0, 48.47, 106.48], [9E9, 9E9, 9E9, 9E9, 9E9, 9E9]];
	VAR jointtarget CDP_1612 := [[10.83, 36.34, 5.2, 0, 48.46, 105.8], [9E9, 9E9, 9E9, 9E9, 9E9, 9E9]];
	VAR jointtarget CDP_1613 := [[10.82, 36.34, 5.2, 0, 48.46, 105.12], [9E9, 9E9, 9E9, 9E9, 9E9, 9E9]];
	VAR jointtarget CDP_1614 := [[10.8, 36.33, 5.21, 0, 48.46, 104.44], [9E9, 9E9, 9E9, 9E9, 9E9, 9E9]];
	VAR jointtarget CDP_1615 := [[10.79, 36.33, 5.22, 0, 48.45, 103.77], [9E9, 9E9, 9E9, 9E9, 9E9, 9E9]];
	VAR jointtarget CDP_1616 := [[10.77, 36.32, 5.23, 0, 48.45, 103.09], [9E9, 9E9, 9E9, 9E9, 9E9, 9E9]];
	VAR jointtarget CDP_1617 := [[10.75, 36.32, 5.23, 0, 48.45, 102.41], [9E9, 9E9, 9E9, 9E9, 9E9, 9E9]];
	VAR jointtarget CDP_1618 := [[10.74, 36.31, 5.24, 0, 48.45, 101.73], [9E9, 9E9, 9E9, 9E9, 9E9, 9E9]];
	VAR jointtarget CDP_1619 := [[10.72, 36.31, 5.25, 0, 48.44, 101.05], [9E9, 9E9, 9E9, 9E9, 9E9, 9E9]];
	VAR jointtarget CDP_1620 := [[9.64, 36.1, 5.61, 0, 48.29, 99.64], [9E9, 9E9, 9E9, 9E9, 9E9, 9E9]];
	VAR jointtarget CDP_1621 := [[8.56, 35.91, 5.93, 0, 48.16, 98.56], [9E9, 9E9, 9E9, 9E9, 9E9, 9E9]];
	VAR jointtarget CDP_1622 := [[7.47, 35.75, 6.22, 0, 48.04, 97.47], [9E9, 9E9, 9E9, 9E9, 9E9, 9E9]];
	VAR jointtarget CDP_1623 := [[6.38, 35.6, 6.46, 0, 47.94, 96.38], [9E9, 9E9, 9E9, 9E9, 9E9, 9E9]];
	VAR jointtarget CDP_1624 := [[5.28, 35.48, 6.67, 0, 47.85, 95.28], [9E9, 9E9, 9E9, 9E9, 9E9, 9E9]];
	VAR jointtarget CDP_1625 := [[4.17, 35.38, 6.83, 0, 47.78, 94.17], [9E9, 9E9, 9E9, 9E9, 9E9, 9E9]];
	VAR jointtarget CDP_1626 := [[3.07, 35.31, 6.96, 0, 47.73, 93.07], [9E9, 9E9, 9E9, 9E9, 9E9, 9E9]];
	VAR jointtarget CDP_1627 := [[1.96, 35.26, 7.05, 0, 47.69, 91.96], [9E9, 9E9, 9E9, 9E9, 9E9, 9E9]];
	VAR jointtarget CDP_1628 := [[0.85, 35.23, 7.1, 0, 47.67, 90.85], [9E9, 9E9, 9E9, 9E9, 9E9, 9E9]];
	VAR jointtarget CDP_1629 := [[-0.26, 35.22, 7.11, 0, 47.67, 89.74], [9E9, 9E9, 9E9, 9E9, 9E9, 9E9]];
	VAR jointtarget CDP_1630 := [[-1.37, 35.24, 7.08, 0, 47.68, 88.63], [9E9, 9E9, 9E9, 9E9, 9E9, 9E9]];
	VAR jointtarget CDP_1631 := [[-2.48, 35.28, 7.01, 0, 47.71, 87.52], [9E9, 9E9, 9E9, 9E9, 9E9, 9E9]];
	VAR jointtarget CDP_1632 := [[-3.59, 35.34, 6.9, 0, 47.75, 86.41], [9E9, 9E9, 9E9, 9E9, 9E9, 9E9]];
	VAR jointtarget CDP_1633 := [[-4.7, 35.43, 6.76, 0, 47.81, 85.3], [9E9, 9E9, 9E9, 9E9, 9E9, 9E9]];
	VAR jointtarget CDP_1634 := [[-5.8, 35.54, 6.57, 0, 47.89, 84.2], [9E9, 9E9, 9E9, 9E9, 9E9, 9E9]];
	VAR jointtarget CDP_1635 := [[-6.9, 35.67, 6.35, 0, 47.98, 83.1], [9E9, 9E9, 9E9, 9E9, 9E9, 9E9]];
	VAR jointtarget CDP_1636 := [[-7.99, 35.82, 6.09, 0, 48.09, 82.01], [9E9, 9E9, 9E9, 9E9, 9E9, 9E9]];
	VAR jointtarget CDP_1637 := [[-9.08, 36, 5.78, 0, 48.22, 80.92], [9E9, 9E9, 9E9, 9E9, 9E9, 9E9]];
	VAR jointtarget CDP_1638 := [[-10.16, 36.2, 5.44, 0, 48.36, 79.84], [9E9, 9E9, 9E9, 9E9, 9E9, 9E9]];
	VAR jointtarget CDP_1639 := [[-11.23, 36.42, 5.06, 0, 48.52, 78.77], [9E9, 9E9, 9E9, 9E9, 9E9, 9E9]];
	VAR jointtarget CDP_1640 := [[-11.28, 36.43, 5.04, 0, 48.53, 79.81], [9E9, 9E9, 9E9, 9E9, 9E9, 9E9]];
	VAR jointtarget CDP_1641 := [[-11.34, 36.44, 5.03, 0, 48.53, 81.95], [9E9, 9E9, 9E9, 9E9, 9E9, 9E9]];
	VAR jointtarget CDP_1642 := [[-11.39, 36.44, 5.02, 0, 48.54, 84.09], [9E9, 9E9, 9E9, 9E9, 9E9, 9E9]];
	VAR jointtarget CDP_1643 := [[-11.45, 36.45, 5.01, 0, 48.54, 86.23], [9E9, 9E9, 9E9, 9E9, 9E9, 9E9]];
	VAR jointtarget CDP_1644 := [[-11.5, 36.45, 5.01, 0, 48.54, 88.37], [9E9, 9E9, 9E9, 9E9, 9E9, 9E9]];
	VAR jointtarget CDP_1645 := [[-11.56, 36.45, 5.01, 0, 48.54, 90.51], [9E9, 9E9, 9E9, 9E9, 9E9, 9E9]];
	VAR jointtarget CDP_1646 := [[-11.61, 36.45, 5.01, 0, 48.54, 92.65], [9E9, 9E9, 9E9, 9E9, 9E9, 9E9]];
	VAR jointtarget CDP_1647 := [[-11.67, 36.44, 5.02, 0, 48.54, 94.78], [9E9, 9E9, 9E9, 9E9, 9E9, 9E9]];
	VAR jointtarget CDP_1648 := [[-11.72, 36.43, 5.03, 0, 48.53, 96.92], [9E9, 9E9, 9E9, 9E9, 9E9, 9E9]];
	VAR jointtarget CDP_1649 := [[-11.78, 36.42, 5.05, 0, 48.52, 99.06], [9E9, 9E9, 9E9, 9E9, 9E9, 9E9]];
	VAR jointtarget CDP_1650 := [[-11.83, 36.41, 5.07, 0, 48.52, 101.2], [9E9, 9E9, 9E9, 9E9, 9E9, 9E9]];
	VAR jointtarget CDP_1651 := [[-11.89, 36.4, 5.1, 0, 48.51, 103.34], [9E9, 9E9, 9E9, 9E9, 9E9, 9E9]];
	VAR jointtarget CDP_1652 := [[-11.94, 36.38, 5.12, 0, 48.49, 105.48], [9E9, 9E9, 9E9, 9E9, 9E9, 9E9]];
	VAR jointtarget CDP_1653 := [[-11.99, 36.36, 5.15, 0, 48.48, 107.63], [9E9, 9E9, 9E9, 9E9, 9E9, 9E9]];
	VAR jointtarget CDP_1654 := [[-12.04, 36.34, 5.19, 0, 48.47, 109.77], [9E9, 9E9, 9E9, 9E9, 9E9, 9E9]];
	VAR jointtarget CDP_1655 := [[-12.09, 36.32, 5.23, 0, 48.45, 111.91], [9E9, 9E9, 9E9, 9E9, 9E9, 9E9]];
	VAR jointtarget CDP_1656 := [[-12.15, 36.3, 5.27, 0, 48.43, 114.05], [9E9, 9E9, 9E9, 9E9, 9E9, 9E9]];
	VAR jointtarget CDP_1657 := [[-12.19, 36.27, 5.32, 0, 48.41, 116.2], [9E9, 9E9, 9E9, 9E9, 9E9, 9E9]];
	VAR jointtarget CDP_1658 := [[-12.24, 36.24, 5.37, 0, 48.39, 118.34], [9E9, 9E9, 9E9, 9E9, 9E9, 9E9]];
	VAR jointtarget CDP_1659 := [[-12.29, 36.21, 5.42, 0, 48.37, 120.49], [9E9, 9E9, 9E9, 9E9, 9E9, 9E9]];
	VAR jointtarget CDP_1660 := [[-12.32, 36.19, 5.45, 0, 48.36, 121.56], [9E9, 9E9, 9E9, 9E9, 9E9, 9E9]];
	VAR jointtarget CDP_1661 := [[-12.35, 36.17, 5.48, 0, 48.34, 121.53], [9E9, 9E9, 9E9, 9E9, 9E9, 9E9]];
	VAR jointtarget CDP_1662 := [[-12.38, 36.15, 5.52, 0, 48.33, 121.5], [9E9, 9E9, 9E9, 9E9, 9E9, 9E9]];
	VAR jointtarget CDP_1663 := [[-12.41, 36.13, 5.55, 0, 48.32, 121.47], [9E9, 9E9, 9E9, 9E9, 9E9, 9E9]];
	VAR jointtarget CDP_1664 := [[-12.43, 36.12, 5.58, 0, 48.3, 121.44], [9E9, 9E9, 9E9, 9E9, 9E9, 9E9]];
	VAR jointtarget CDP_1665 := [[-12.46, 36.1, 5.61, 0, 48.29, 121.41], [9E9, 9E9, 9E9, 9E9, 9E9, 9E9]];
	VAR jointtarget CDP_1666 := [[-12.49, 36.08, 5.65, 0, 48.28, 121.39], [9E9, 9E9, 9E9, 9E9, 9E9, 9E9]];
	VAR jointtarget CDP_1667 := [[-12.52, 36.06, 5.68, 0, 48.26, 121.36], [9E9, 9E9, 9E9, 9E9, 9E9, 9E9]];
	VAR jointtarget CDP_1668 := [[-12.55, 36.04, 5.71, 0, 48.25, 121.33], [9E9, 9E9, 9E9, 9E9, 9E9, 9E9]];
	VAR jointtarget CDP_1669 := [[-12.58, 36.02, 5.75, 0, 48.23, 121.3], [9E9, 9E9, 9E9, 9E9, 9E9, 9E9]];
	VAR jointtarget CDP_1670 := [[-12.61, 36, 5.78, 0, 48.22, 121.27], [9E9, 9E9, 9E9, 9E9, 9E9, 9E9]];
	VAR jointtarget CDP_1671 := [[-12.63, 35.98, 5.81, 0, 48.21, 121.24], [9E9, 9E9, 9E9, 9E9, 9E9, 9E9]];
	VAR jointtarget CDP_1672 := [[-12.66, 35.96, 5.84, 0, 48.19, 121.21], [9E9, 9E9, 9E9, 9E9, 9E9, 9E9]];
	VAR jointtarget CDP_1673 := [[-12.69, 35.94, 5.87, 0, 48.18, 121.18], [9E9, 9E9, 9E9, 9E9, 9E9, 9E9]];
	VAR jointtarget CDP_1674 := [[-12.72, 35.93, 5.91, 0, 48.17, 121.16], [9E9, 9E9, 9E9, 9E9, 9E9, 9E9]];
	VAR jointtarget CDP_1675 := [[-12.75, 35.91, 5.94, 0, 48.15, 121.13], [9E9, 9E9, 9E9, 9E9, 9E9, 9E9]];
	VAR jointtarget CDP_1676 := [[-12.78, 35.89, 5.97, 0, 48.14, 121.1], [9E9, 9E9, 9E9, 9E9, 9E9, 9E9]];
	VAR jointtarget CDP_1677 := [[-12.81, 35.87, 6, 0, 48.13, 121.07], [9E9, 9E9, 9E9, 9E9, 9E9, 9E9]];
	VAR jointtarget CDP_1678 := [[-12.84, 35.85, 6.04, 0, 48.11, 121.04], [9E9, 9E9, 9E9, 9E9, 9E9, 9E9]];
	VAR jointtarget CDP_1679 := [[-12.86, 35.83, 6.07, 0, 48.1, 121.01], [9E9, 9E9, 9E9, 9E9, 9E9, 9E9]];
	VAR jointtarget CDP_1680 := [[-13.02, 35.76, 6.19, 0, 48.05, 114.17], [9E9, 9E9, 9E9, 9E9, 9E9, 9E9]];
	VAR jointtarget CDP_1681 := [[-13.18, 35.73, 6.25, 0, 48.02, 100.62], [9E9, 9E9, 9E9, 9E9, 9E9, 9E9]];
	VAR jointtarget CDP_1682 := [[-13.34, 35.73, 6.23, 0, 48.03, 87.07], [9E9, 9E9, 9E9, 9E9, 9E9, 9E9]];
	VAR jointtarget CDP_1683 := [[-13.5, 35.79, 6.15, 0, 48.07, 73.52], [9E9, 9E9, 9E9, 9E9, 9E9, 9E9]];
	VAR jointtarget CDP_1684 := [[-13.64, 35.87, 6, 0, 48.13, 59.99], [9E9, 9E9, 9E9, 9E9, 9E9, 9E9]];
	VAR jointtarget CDP_1685 := [[-13.76, 36, 5.79, 0, 48.22, 46.48], [9E9, 9E9, 9E9, 9E9, 9E9, 9E9]];
	VAR jointtarget CDP_1686 := [[-13.85, 36.15, 5.53, 0, 48.32, 33.01], [9E9, 9E9, 9E9, 9E9, 9E9, 9E9]];
	VAR jointtarget CDP_1687 := [[-13.91, 36.31, 5.24, 0, 48.44, 19.56], [9E9, 9E9, 9E9, 9E9, 9E9, 9E9]];
	VAR jointtarget CDP_1688 := [[-13.92, 36.49, 4.94, 0, 48.57, 6.16], [9E9, 9E9, 9E9, 9E9, 9E9, 9E9]];
	VAR jointtarget CDP_1689 := [[-13.9, 36.67, 4.63, 0, 48.7, -7.21], [9E9, 9E9, 9E9, 9E9, 9E9, 9E9]];
	VAR jointtarget CDP_1690 := [[-13.85, 36.84, 4.34, 0, 48.82, -20.54], [9E9, 9E9, 9E9, 9E9, 9E9, 9E9]];
	VAR jointtarget CDP_1691 := [[-13.76, 36.99, 4.08, 0, 48.93, -33.84], [9E9, 9E9, 9E9, 9E9, 9E9, 9E9]];
	VAR jointtarget CDP_1692 := [[-13.64, 37.11, 3.87, 0, 49.02, -47.11], [9E9, 9E9, 9E9, 9E9, 9E9, 9E9]];
	VAR jointtarget CDP_1693 := [[-13.5, 37.2, 3.72, 0, 49.08, -60.35], [9E9, 9E9, 9E9, 9E9, 9E9, 9E9]];
	VAR jointtarget CDP_1694 := [[-13.34, 37.25, 3.63, 0, 49.12, -73.59], [9E9, 9E9, 9E9, 9E9, 9E9, 9E9]];
	VAR jointtarget CDP_1695 := [[-13.18, 37.26, 3.62, 0, 49.13, -86.81], [9E9, 9E9, 9E9, 9E9, 9E9, 9E9]];
	VAR jointtarget CDP_1696 := [[-13.02, 37.23, 3.67, 0, 49.1, -100.04], [9E9, 9E9, 9E9, 9E9, 9E9, 9E9]];
	VAR jointtarget CDP_1697 := [[-12.88, 37.15, 3.79, 0, 49.05, -113.28], [9E9, 9E9, 9E9, 9E9, 9E9, 9E9]];
	VAR jointtarget CDP_1698 := [[-12.75, 37.05, 3.98, 0, 48.97, -126.54], [9E9, 9E9, 9E9, 9E9, 9E9, 9E9]];
	VAR jointtarget CDP_1699 := [[-12.64, 36.91, 4.22, 0, 48.87, -139.82], [9E9, 9E9, 9E9, 9E9, 9E9, 9E9]];
	VAR jointtarget CDP_1700 := [[-12.62, 36.87, 4.29, 0, 48.84, -146.49], [9E9, 9E9, 9E9, 9E9, 9E9, 9E9]];
	VAR jointtarget CDP_1701 := [[-12.59, 36.83, 4.36, 0, 48.81, -146.47], [9E9, 9E9, 9E9, 9E9, 9E9, 9E9]];
	VAR jointtarget CDP_1702 := [[-12.57, 36.79, 4.43, 0, 48.78, -146.44], [9E9, 9E9, 9E9, 9E9, 9E9, 9E9]];
	VAR jointtarget CDP_1703 := [[-12.54, 36.75, 4.5, 0, 48.76, -146.42], [9E9, 9E9, 9E9, 9E9, 9E9, 9E9]];
	VAR jointtarget CDP_1704 := [[-12.52, 36.7, 4.57, 0, 48.73, -146.4], [9E9, 9E9, 9E9, 9E9, 9E9, 9E9]];
	VAR jointtarget CDP_1705 := [[-12.49, 36.66, 4.64, 0, 48.7, -146.37], [9E9, 9E9, 9E9, 9E9, 9E9, 9E9]];
	VAR jointtarget CDP_1706 := [[-12.47, 36.62, 4.71, 0, 48.67, -146.35], [9E9, 9E9, 9E9, 9E9, 9E9, 9E9]];
	VAR jointtarget CDP_1707 := [[-12.44, 36.58, 4.78, 0, 48.64, -146.32], [9E9, 9E9, 9E9, 9E9, 9E9, 9E9]];
	VAR jointtarget CDP_1708 := [[-12.42, 36.54, 4.85, 0, 48.61, -146.3], [9E9, 9E9, 9E9, 9E9, 9E9, 9E9]];
	VAR jointtarget CDP_1709 := [[-12.39, 36.5, 4.92, 0, 48.58, -146.27], [9E9, 9E9, 9E9, 9E9, 9E9, 9E9]];
	VAR jointtarget CDP_1710 := [[-12.37, 36.46, 4.99, 0, 48.55, -146.25], [9E9, 9E9, 9E9, 9E9, 9E9, 9E9]];
	VAR jointtarget CDP_1711 := [[-12.34, 36.42, 5.06, 0, 48.52, -146.22], [9E9, 9E9, 9E9, 9E9, 9E9, 9E9]];
	VAR jointtarget CDP_1712 := [[-12.32, 36.38, 5.13, 0, 48.49, -146.2], [9E9, 9E9, 9E9, 9E9, 9E9, 9E9]];
	VAR jointtarget CDP_1713 := [[-12.29, 36.34, 5.2, 0, 48.46, -146.17], [9E9, 9E9, 9E9, 9E9, 9E9, 9E9]];
	VAR jointtarget CDP_1714 := [[-12.27, 36.29, 5.27, 0, 48.43, -146.15], [9E9, 9E9, 9E9, 9E9, 9E9, 9E9]];
	VAR jointtarget CDP_1715 := [[-12.24, 36.25, 5.34, 0, 48.4, -146.12], [9E9, 9E9, 9E9, 9E9, 9E9, 9E9]];
	VAR jointtarget CDP_1716 := [[-12.22, 36.21, 5.41, 0, 48.37, -146.1], [9E9, 9E9, 9E9, 9E9, 9E9, 9E9]];
	VAR jointtarget CDP_1717 := [[-12.19, 36.17, 5.48, 0, 48.34, -146.07], [9E9, 9E9, 9E9, 9E9, 9E9, 9E9]];
	VAR jointtarget CDP_1718 := [[-12.17, 36.13, 5.55, 0, 48.31, -146.05], [9E9, 9E9, 9E9, 9E9, 9E9, 9E9]];
	VAR jointtarget CDP_1719 := [[-12.14, 36.09, 5.62, 0, 48.28, -146.02], [9E9, 9E9, 9E9, 9E9, 9E9, 9E9]];
	VAR jointtarget CDP_1720 := [[-12.14, 36.08, 5.65, 0, 48.28, -145.46], [9E9, 9E9, 9E9, 9E9, 9E9, 9E9]];
	VAR jointtarget CDP_1721 := [[-12.13, 36.07, 5.67, 0, 48.27, -144.35], [9E9, 9E9, 9E9, 9E9, 9E9, 9E9]];
	VAR jointtarget CDP_1722 := [[-12.12, 36.05, 5.69, 0, 48.26, -143.24], [9E9, 9E9, 9E9, 9E9, 9E9, 9E9]];
	VAR jointtarget CDP_1723 := [[-12.11, 36.04, 5.71, 0, 48.25, -142.13], [9E9, 9E9, 9E9, 9E9, 9E9, 9E9]];
	VAR jointtarget CDP_1724 := [[-12.1, 36.03, 5.73, 0, 48.24, -141.01], [9E9, 9E9, 9E9, 9E9, 9E9, 9E9]];
	VAR jointtarget CDP_1725 := [[-12.09, 36.02, 5.75, 0, 48.23, -139.9], [9E9, 9E9, 9E9, 9E9, 9E9, 9E9]];
	VAR jointtarget CDP_1726 := [[-12.08, 36.01, 5.77, 0, 48.23, -138.79], [9E9, 9E9, 9E9, 9E9, 9E9, 9E9]];
	VAR jointtarget CDP_1727 := [[-12.07, 35.99, 5.79, 0, 48.22, -137.68], [9E9, 9E9, 9E9, 9E9, 9E9, 9E9]];
	VAR jointtarget CDP_1728 := [[-12.06, 35.98, 5.81, 0, 48.21, -136.56], [9E9, 9E9, 9E9, 9E9, 9E9, 9E9]];
	VAR jointtarget CDP_1729 := [[-12.05, 35.97, 5.83, 0, 48.2, -135.45], [9E9, 9E9, 9E9, 9E9, 9E9, 9E9]];
	VAR jointtarget CDP_1730 := [[-12.04, 35.96, 5.84, 0, 48.19, -134.34], [9E9, 9E9, 9E9, 9E9, 9E9, 9E9]];
	VAR jointtarget CDP_1731 := [[-12.03, 35.95, 5.86, 0, 48.19, -133.22], [9E9, 9E9, 9E9, 9E9, 9E9, 9E9]];
	VAR jointtarget CDP_1732 := [[-12.02, 35.94, 5.88, 0, 48.18, -132.11], [9E9, 9E9, 9E9, 9E9, 9E9, 9E9]];
	VAR jointtarget CDP_1733 := [[-12.01, 35.93, 5.9, 0, 48.17, -130.99], [9E9, 9E9, 9E9, 9E9, 9E9, 9E9]];
	VAR jointtarget CDP_1734 := [[-12, 35.92, 5.91, 0, 48.17, -129.88], [9E9, 9E9, 9E9, 9E9, 9E9, 9E9]];
	VAR jointtarget CDP_1735 := [[-11.99, 35.91, 5.93, 0, 48.16, -128.76], [9E9, 9E9, 9E9, 9E9, 9E9, 9E9]];
	VAR jointtarget CDP_1736 := [[-11.98, 35.9, 5.94, 0, 48.16, -127.65], [9E9, 9E9, 9E9, 9E9, 9E9, 9E9]];
	VAR jointtarget CDP_1737 := [[-11.97, 35.89, 5.96, 0, 48.15, -126.53], [9E9, 9E9, 9E9, 9E9, 9E9, 9E9]];
	VAR jointtarget CDP_1738 := [[-11.96, 35.88, 5.98, 0, 48.14, -125.42], [9E9, 9E9, 9E9, 9E9, 9E9, 9E9]];
	VAR jointtarget CDP_1739 := [[-11.95, 35.87, 5.99, 0, 48.14, -124.3], [9E9, 9E9, 9E9, 9E9, 9E9, 9E9]];
	VAR jointtarget CDP_1740 := [[-11.94, 35.86, 6, 0, 48.13, -123.74], [9E9, 9E9, 9E9, 9E9, 9E9, 9E9]];
	VAR jointtarget CDP_1741 := [[-11.93, 35.86, 6.02, 0, 48.13, -123.73], [9E9, 9E9, 9E9, 9E9, 9E9, 9E9]];
	VAR jointtarget CDP_1742 := [[-11.92, 35.85, 6.03, 0, 48.12, -123.72], [9E9, 9E9, 9E9, 9E9, 9E9, 9E9]];
	VAR jointtarget CDP_1743 := [[-11.9, 35.84, 6.04, 0, 48.12, -123.71], [9E9, 9E9, 9E9, 9E9, 9E9, 9E9]];
	VAR jointtarget CDP_1744 := [[-11.89, 35.83, 6.05, 0, 48.11, -123.7], [9E9, 9E9, 9E9, 9E9, 9E9, 9E9]];
	VAR jointtarget CDP_1745 := [[-11.88, 35.82, 6.07, 0, 48.11, -123.69], [9E9, 9E9, 9E9, 9E9, 9E9, 9E9]];
	VAR jointtarget CDP_1746 := [[-11.87, 35.82, 6.08, 0, 48.1, -123.68], [9E9, 9E9, 9E9, 9E9, 9E9, 9E9]];
	VAR jointtarget CDP_1747 := [[-11.86, 35.81, 6.09, 0, 48.1, -123.66], [9E9, 9E9, 9E9, 9E9, 9E9, 9E9]];
	VAR jointtarget CDP_1748 := [[-11.85, 35.8, 6.1, 0, 48.09, -123.65], [9E9, 9E9, 9E9, 9E9, 9E9, 9E9]];
	VAR jointtarget CDP_1749 := [[-11.84, 35.79, 6.12, 0, 48.09, -123.64], [9E9, 9E9, 9E9, 9E9, 9E9, 9E9]];
	VAR jointtarget CDP_1750 := [[-11.83, 35.79, 6.13, 0, 48.08, -123.63], [9E9, 9E9, 9E9, 9E9, 9E9, 9E9]];
	VAR jointtarget CDP_1751 := [[-11.82, 35.78, 6.14, 0, 48.08, -123.62], [9E9, 9E9, 9E9, 9E9, 9E9, 9E9]];
	VAR jointtarget CDP_1752 := [[-11.81, 35.77, 6.16, 0, 48.08, -123.61], [9E9, 9E9, 9E9, 9E9, 9E9, 9E9]];
	VAR jointtarget CDP_1753 := [[-11.8, 35.76, 6.17, 0, 48.07, -123.6], [9E9, 9E9, 9E9, 9E9, 9E9, 9E9]];
	VAR jointtarget CDP_1754 := [[-11.79, 35.75, 6.18, 0, 48.07, -123.59], [9E9, 9E9, 9E9, 9E9, 9E9, 9E9]];
	VAR jointtarget CDP_1755 := [[-11.78, 35.75, 6.19, 0, 48.06, -123.58], [9E9, 9E9, 9E9, 9E9, 9E9, 9E9]];
	VAR jointtarget CDP_1756 := [[-11.77, 35.74, 6.21, 0, 48.06, -123.57], [9E9, 9E9, 9E9, 9E9, 9E9, 9E9]];
	VAR jointtarget CDP_1757 := [[-11.76, 35.73, 6.22, 0, 48.05, -123.56], [9E9, 9E9, 9E9, 9E9, 9E9, 9E9]];
	VAR jointtarget CDP_1758 := [[-11.75, 35.72, 6.23, 0, 48.05, -123.55], [9E9, 9E9, 9E9, 9E9, 9E9, 9E9]];
	VAR jointtarget CDP_1759 := [[-11.74, 35.71, 6.24, 0, 48.04, -123.54], [9E9, 9E9, 9E9, 9E9, 9E9, 9E9]];
	VAR jointtarget CDP_1760 := [[-10.65, 35.48, 6.64, 0, 47.88, -100.65], [9E9, 9E9, 9E9, 9E9, 9E9, 9E9]];
	VAR jointtarget CDP_1761 := [[-9.55, 35.27, 7, 0, 47.73, -99.55], [9E9, 9E9, 9E9, 9E9, 9E9, 9E9]];
	VAR jointtarget CDP_1762 := [[-8.44, 35.09, 7.32, 0, 47.6, -98.44], [9E9, 9E9, 9E9, 9E9, 9E9, 9E9]];
	VAR jointtarget CDP_1763 := [[-7.33, 34.92, 7.6, 0, 47.48, -97.33], [9E9, 9E9, 9E9, 9E9, 9E9, 9E9]];
	VAR jointtarget CDP_1764 := [[-6.21, 34.78, 7.83, 0, 47.38, -96.21], [9E9, 9E9, 9E9, 9E9, 9E9, 9E9]];
	VAR jointtarget CDP_1765 := [[-5.09, 34.67, 8.03, 0, 47.3, -95.09], [9E9, 9E9, 9E9, 9E9, 9E9, 9E9]];
	VAR jointtarget CDP_1766 := [[-3.96, 34.57, 8.19, 0, 47.24, -93.96], [9E9, 9E9, 9E9, 9E9, 9E9, 9E9]];
	VAR jointtarget CDP_1767 := [[-2.83, 34.5, 8.31, 0, 47.19, -92.83], [9E9, 9E9, 9E9, 9E9, 9E9, 9E9]];
	VAR jointtarget CDP_1768 := [[-1.7, 34.46, 8.39, 0, 47.15, -91.7], [9E9, 9E9, 9E9, 9E9, 9E9, 9E9]];
	VAR jointtarget CDP_1769 := [[-0.56, 34.43, 8.43, 0, 47.14, -90.56], [9E9, 9E9, 9E9, 9E9, 9E9, 9E9]];
	VAR jointtarget CDP_1770 := [[0.57, 34.43, 8.43, 0, 47.14, -89.43], [9E9, 9E9, 9E9, 9E9, 9E9, 9E9]];
	VAR jointtarget CDP_1771 := [[1.7, 34.46, 8.39, 0, 47.15, -88.3], [9E9, 9E9, 9E9, 9E9, 9E9, 9E9]];
	VAR jointtarget CDP_1772 := [[2.84, 34.5, 8.31, 0, 47.19, -87.16], [9E9, 9E9, 9E9, 9E9, 9E9, 9E9]];
	VAR jointtarget CDP_1773 := [[3.97, 34.57, 8.19, 0, 47.24, -86.03], [9E9, 9E9, 9E9, 9E9, 9E9, 9E9]];
	VAR jointtarget CDP_1774 := [[5.09, 34.67, 8.03, 0, 47.3, -84.91], [9E9, 9E9, 9E9, 9E9, 9E9, 9E9]];
	VAR jointtarget CDP_1775 := [[6.22, 34.78, 7.83, 0, 47.38, -83.78], [9E9, 9E9, 9E9, 9E9, 9E9, 9E9]];
	VAR jointtarget CDP_1776 := [[7.34, 34.92, 7.59, 0, 47.48, -82.66], [9E9, 9E9, 9E9, 9E9, 9E9, 9E9]];
	VAR jointtarget CDP_1777 := [[8.45, 35.09, 7.31, 0, 47.6, -81.55], [9E9, 9E9, 9E9, 9E9, 9E9, 9E9]];
	VAR jointtarget CDP_1778 := [[9.56, 35.27, 7, 0, 47.73, -80.44], [9E9, 9E9, 9E9, 9E9, 9E9, 9E9]];
	VAR jointtarget CDP_1779 := [[10.65, 35.48, 6.64, 0, 47.88, -79.35], [9E9, 9E9, 9E9, 9E9, 9E9, 9E9]];
	VAR jointtarget CDP_1780 := [[10.71, 35.5, 6.62, 0, 47.89, -78.19], [9E9, 9E9, 9E9, 9E9, 9E9, 9E9]];
	VAR jointtarget CDP_1781 := [[10.76, 35.51, 6.59, 0, 47.9, -75.95], [9E9, 9E9, 9E9, 9E9, 9E9, 9E9]];
	VAR jointtarget CDP_1782 := [[10.82, 35.53, 6.56, 0, 47.91, -73.7], [9E9, 9E9, 9E9, 9E9, 9E9, 9E9]];
	VAR jointtarget CDP_1783 := [[10.87, 35.55, 6.53, 0, 47.92, -71.45], [9E9, 9E9, 9E9, 9E9, 9E9, 9E9]];
	VAR jointtarget CDP_1784 := [[10.92, 35.57, 6.49, 0, 47.94, -69.2], [9E9, 9E9, 9E9, 9E9, 9E9, 9E9]];
	VAR jointtarget CDP_1785 := [[10.97, 35.59, 6.45, 0, 47.95, -66.96], [9E9, 9E9, 9E9, 9E9, 9E9, 9E9]];
	VAR jointtarget CDP_1786 := [[11.03, 35.62, 6.41, 0, 47.97, -64.72], [9E9, 9E9, 9E9, 9E9, 9E9, 9E9]];
	VAR jointtarget CDP_1787 := [[11.07, 35.64, 6.36, 0, 47.99, -62.47], [9E9, 9E9, 9E9, 9E9, 9E9, 9E9]];
	VAR jointtarget CDP_1788 := [[11.12, 35.67, 6.31, 0, 48.01, -60.23], [9E9, 9E9, 9E9, 9E9, 9E9, 9E9]];
	VAR jointtarget CDP_1789 := [[11.17, 35.71, 6.26, 0, 48.04, -57.99], [9E9, 9E9, 9E9, 9E9, 9E9, 9E9]];
	VAR jointtarget CDP_1790 := [[11.22, 35.74, 6.2, 0, 48.06, -55.75], [9E9, 9E9, 9E9, 9E9, 9E9, 9E9]];
	VAR jointtarget CDP_1791 := [[11.26, 35.78, 6.14, 0, 48.09, -53.51], [9E9, 9E9, 9E9, 9E9, 9E9, 9E9]];
	VAR jointtarget CDP_1792 := [[11.3, 35.81, 6.07, 0, 48.11, -51.27], [9E9, 9E9, 9E9, 9E9, 9E9, 9E9]];
	VAR jointtarget CDP_1793 := [[11.35, 35.85, 6.01, 0, 48.14, -49.04], [9E9, 9E9, 9E9, 9E9, 9E9, 9E9]];
	VAR jointtarget CDP_1794 := [[11.39, 35.89, 5.94, 0, 48.17, -46.8], [9E9, 9E9, 9E9, 9E9, 9E9, 9E9]];
	VAR jointtarget CDP_1795 := [[11.43, 35.94, 5.86, 0, 48.2, -44.57], [9E9, 9E9, 9E9, 9E9, 9E9, 9E9]];
	VAR jointtarget CDP_1796 := [[11.46, 35.98, 5.79, 0, 48.23, -42.34], [9E9, 9E9, 9E9, 9E9, 9E9, 9E9]];
	VAR jointtarget CDP_1797 := [[11.5, 36.03, 5.71, 0, 48.26, -40.11], [9E9, 9E9, 9E9, 9E9, 9E9, 9E9]];
	VAR jointtarget CDP_1798 := [[11.53, 36.08, 5.63, 0, 48.3, -37.88], [9E9, 9E9, 9E9, 9E9, 9E9, 9E9]];
	VAR jointtarget CDP_1799 := [[11.57, 36.12, 5.54, 0, 48.33, -35.65], [9E9, 9E9, 9E9, 9E9, 9E9, 9E9]];
	VAR jointtarget CDP_1800 := [[11.59, 36.15, 5.49, 0, 48.36, -34.54], [9E9, 9E9, 9E9, 9E9, 9E9, 9E9]];
	VAR jointtarget CDP_1801 := [[11.6, 36.18, 5.44, 0, 48.38, -34.52], [9E9, 9E9, 9E9, 9E9, 9E9, 9E9]];
	VAR jointtarget CDP_1802 := [[11.62, 36.21, 5.39, 0, 48.4, -34.5], [9E9, 9E9, 9E9, 9E9, 9E9, 9E9]];
	VAR jointtarget CDP_1803 := [[11.64, 36.24, 5.34, 0, 48.42, -34.48], [9E9, 9E9, 9E9, 9E9, 9E9, 9E9]];
	VAR jointtarget CDP_1804 := [[11.66, 36.28, 5.28, 0, 48.44, -34.46], [9E9, 9E9, 9E9, 9E9, 9E9, 9E9]];
	VAR jointtarget CDP_1805 := [[11.68, 36.31, 5.23, 0, 48.46, -34.44], [9E9, 9E9, 9E9, 9E9, 9E9, 9E9]];
	VAR jointtarget CDP_1806 := [[11.7, 36.34, 5.18, 0, 48.48, -34.42], [9E9, 9E9, 9E9, 9E9, 9E9, 9E9]];
	VAR jointtarget CDP_1807 := [[11.72, 36.37, 5.13, 0, 48.51, -34.41], [9E9, 9E9, 9E9, 9E9, 9E9, 9E9]];
	VAR jointtarget CDP_1808 := [[11.74, 36.4, 5.08, 0, 48.53, -34.39], [9E9, 9E9, 9E9, 9E9, 9E9, 9E9]];
	VAR jointtarget CDP_1809 := [[11.76, 36.43, 5.02, 0, 48.55, -34.37], [9E9, 9E9, 9E9, 9E9, 9E9, 9E9]];
	VAR jointtarget CDP_1810 := [[11.77, 36.46, 4.97, 0, 48.57, -34.35], [9E9, 9E9, 9E9, 9E9, 9E9, 9E9]];
	VAR jointtarget CDP_1811 := [[11.79, 36.49, 4.92, 0, 48.59, -34.33], [9E9, 9E9, 9E9, 9E9, 9E9, 9E9]];
	VAR jointtarget CDP_1812 := [[11.81, 36.52, 4.87, 0, 48.61, -34.31], [9E9, 9E9, 9E9, 9E9, 9E9, 9E9]];
	VAR jointtarget CDP_1813 := [[11.83, 36.55, 4.82, 0, 48.64, -34.29], [9E9, 9E9, 9E9, 9E9, 9E9, 9E9]];
	VAR jointtarget CDP_1814 := [[11.85, 36.58, 4.76, 0, 48.66, -34.27], [9E9, 9E9, 9E9, 9E9, 9E9, 9E9]];
	VAR jointtarget CDP_1815 := [[11.87, 36.61, 4.71, 0, 48.68, -34.26], [9E9, 9E9, 9E9, 9E9, 9E9, 9E9]];
	VAR jointtarget CDP_1816 := [[11.89, 36.64, 4.66, 0, 48.7, -34.24], [9E9, 9E9, 9E9, 9E9, 9E9, 9E9]];
	VAR jointtarget CDP_1817 := [[11.91, 36.67, 4.61, 0, 48.72, -34.22], [9E9, 9E9, 9E9, 9E9, 9E9, 9E9]];
	VAR jointtarget CDP_1818 := [[11.92, 36.7, 4.56, 0, 48.75, -34.2], [9E9, 9E9, 9E9, 9E9, 9E9, 9E9]];
	VAR jointtarget CDP_1819 := [[11.94, 36.73, 4.5, 0, 48.77, -34.18], [9E9, 9E9, 9E9, 9E9, 9E9, 9E9]];
	VAR jointtarget CDP_1820 := [[12.05, 36.86, 4.27, 0, 48.87, -40.77], [9E9, 9E9, 9E9, 9E9, 9E9, 9E9]];
	VAR jointtarget CDP_1821 := [[12.18, 36.97, 4.09, 0, 48.94, -54.03], [9E9, 9E9, 9E9, 9E9, 9E9, 9E9]];
	VAR jointtarget CDP_1822 := [[12.33, 37.04, 3.97, 0, 48.99, -67.26], [9E9, 9E9, 9E9, 9E9, 9E9, 9E9]];
	VAR jointtarget CDP_1823 := [[12.49, 37.07, 3.92, 0, 49.01, -80.49], [9E9, 9E9, 9E9, 9E9, 9E9, 9E9]];
	VAR jointtarget CDP_1824 := [[12.65, 37.06, 3.94, 0, 49, -93.72], [9E9, 9E9, 9E9, 9E9, 9E9, 9E9]];
	VAR jointtarget CDP_1825 := [[12.8, 37, 4.03, 0, 48.97, -106.95], [9E9, 9E9, 9E9, 9E9, 9E9, 9E9]];
	VAR jointtarget CDP_1826 := [[12.94, 36.91, 4.19, 0, 48.9, -120.2], [9E9, 9E9, 9E9, 9E9, 9E9, 9E9]];
	VAR jointtarget CDP_1827 := [[13.06, 36.79, 4.4, 0, 48.81, -133.47], [9E9, 9E9, 9E9, 9E9, 9E9, 9E9]];
	VAR jointtarget CDP_1828 := [[13.15, 36.64, 4.66, 0, 48.7, -146.77], [9E9, 9E9, 9E9, 9E9, 9E9, 9E9]];
	VAR jointtarget CDP_1829 := [[13.2, 36.47, 4.95, 0, 48.58, -160.1], [9E9, 9E9, 9E9, 9E9, 9E9, 9E9]];
	VAR jointtarget CDP_1830 := [[13.22, 36.29, 5.25, 0, 48.45, -173.47], [9E9, 9E9, 9E9, 9E9, 9E9, 9E9]];
	VAR jointtarget CDP_1831 := [[13.2, 36.12, 5.56, 0, 48.33, -186.88], [9E9, 9E9, 9E9, 9E9, 9E9, 9E9]];
	VAR jointtarget CDP_1832 := [[13.15, 35.95, 5.84, 0, 48.21, -200.32], [9E9, 9E9, 9E9, 9E9, 9E9, 9E9]];
	VAR jointtarget CDP_1833 := [[13.06, 35.8, 6.1, 0, 48.1, -213.8], [9E9, 9E9, 9E9, 9E9, 9E9, 9E9]];
	VAR jointtarget CDP_1834 := [[12.93, 35.68, 6.3, 0, 48.02, -227.31], [9E9, 9E9, 9E9, 9E9, 9E9, 9E9]];
	VAR jointtarget CDP_1835 := [[12.79, 35.59, 6.45, 0, 47.96, -240.84], [9E9, 9E9, 9E9, 9E9, 9E9, 9E9]];
	VAR jointtarget CDP_1836 := [[12.63, 35.55, 6.53, 0, 47.92, -254.39], [9E9, 9E9, 9E9, 9E9, 9E9, 9E9]];
	VAR jointtarget CDP_1837 := [[12.47, 35.54, 6.54, 0, 47.92, -267.94], [9E9, 9E9, 9E9, 9E9, 9E9, 9E9]];
	VAR jointtarget CDP_1838 := [[12.3, 35.57, 6.48, 0, 47.94, -281.49], [9E9, 9E9, 9E9, 9E9, 9E9, 9E9]];
	VAR jointtarget CDP_1839 := [[12.15, 35.65, 6.36, 0, 47.99, -295.03], [9E9, 9E9, 9E9, 9E9, 9E9, 9E9]];
	VAR jointtarget CDP_1840 := [[12.13, 35.67, 6.32, 0, 48.01, -301.75], [9E9, 9E9, 9E9, 9E9, 9E9, 9E9]];
	VAR jointtarget CDP_1841 := [[12.1, 35.69, 6.29, 0, 48.02, -301.78], [9E9, 9E9, 9E9, 9E9, 9E9, 9E9]];
	VAR jointtarget CDP_1842 := [[12.07, 35.71, 6.26, 0, 48.04, -301.81], [9E9, 9E9, 9E9, 9E9, 9E9, 9E9]];
	VAR jointtarget CDP_1843 := [[12.04, 35.73, 6.23, 0, 48.05, -301.84], [9E9, 9E9, 9E9, 9E9, 9E9, 9E9]];
	VAR jointtarget CDP_1844 := [[12.01, 35.74, 6.19, 0, 48.06, -301.87], [9E9, 9E9, 9E9, 9E9, 9E9, 9E9]];
	VAR jointtarget CDP_1845 := [[11.98, 35.76, 6.16, 0, 48.08, -301.89], [9E9, 9E9, 9E9, 9E9, 9E9, 9E9]];
	VAR jointtarget CDP_1846 := [[11.95, 35.78, 6.13, 0, 48.09, -301.92], [9E9, 9E9, 9E9, 9E9, 9E9, 9E9]];
	VAR jointtarget CDP_1847 := [[11.92, 35.8, 6.09, 0, 48.1, -301.95], [9E9, 9E9, 9E9, 9E9, 9E9, 9E9]];
	VAR jointtarget CDP_1848 := [[11.9, 35.82, 6.06, 0, 48.12, -301.98], [9E9, 9E9, 9E9, 9E9, 9E9, 9E9]];
	VAR jointtarget CDP_1849 := [[11.87, 35.84, 6.03, 0, 48.13, -302.01], [9E9, 9E9, 9E9, 9E9, 9E9, 9E9]];
	VAR jointtarget CDP_1850 := [[11.84, 35.86, 6, 0, 48.14, -302.04], [9E9, 9E9, 9E9, 9E9, 9E9, 9E9]];
	VAR jointtarget CDP_1851 := [[11.81, 35.88, 5.96, 0, 48.16, -302.07], [9E9, 9E9, 9E9, 9E9, 9E9, 9E9]];
	VAR jointtarget CDP_1852 := [[11.78, 35.9, 5.93, 0, 48.17, -302.09], [9E9, 9E9, 9E9, 9E9, 9E9, 9E9]];
	VAR jointtarget CDP_1853 := [[11.75, 35.92, 5.9, 0, 48.19, -302.12], [9E9, 9E9, 9E9, 9E9, 9E9, 9E9]];
	VAR jointtarget CDP_1854 := [[11.73, 35.94, 5.86, 0, 48.2, -302.15], [9E9, 9E9, 9E9, 9E9, 9E9, 9E9]];
	VAR jointtarget CDP_1855 := [[11.7, 35.96, 5.83, 0, 48.21, -302.18], [9E9, 9E9, 9E9, 9E9, 9E9, 9E9]];
	VAR jointtarget CDP_1856 := [[11.67, 35.98, 5.8, 0, 48.23, -302.21], [9E9, 9E9, 9E9, 9E9, 9E9, 9E9]];
	VAR jointtarget CDP_1857 := [[11.64, 36, 5.76, 0, 48.24, -302.24], [9E9, 9E9, 9E9, 9E9, 9E9, 9E9]];
	VAR jointtarget CDP_1858 := [[11.61, 36.02, 5.73, 0, 48.26, -302.27], [9E9, 9E9, 9E9, 9E9, 9E9, 9E9]];
	VAR jointtarget CDP_1859 := [[11.58, 36.03, 5.7, 0, 48.27, -302.29], [9E9, 9E9, 9E9, 9E9, 9E9, 9E9]];
	VAR jointtarget CDP_1860 := [[11.54, 36.07, 5.64, 0, 48.29, -301.24], [9E9, 9E9, 9E9, 9E9, 9E9, 9E9]];
	VAR jointtarget CDP_1861 := [[11.49, 36.1, 5.59, 0, 48.31, -299.1], [9E9, 9E9, 9E9, 9E9, 9E9, 9E9]];
	VAR jointtarget CDP_1862 := [[11.44, 36.12, 5.55, 0, 48.33, -296.95], [9E9, 9E9, 9E9, 9E9, 9E9, 9E9]];
	VAR jointtarget CDP_1863 := [[11.39, 36.15, 5.5, 0, 48.35, -294.81], [9E9, 9E9, 9E9, 9E9, 9E9, 9E9]];
	VAR jointtarget CDP_1864 := [[11.34, 36.17, 5.46, 0, 48.37, -292.67], [9E9, 9E9, 9E9, 9E9, 9E9, 9E9]];
	VAR jointtarget CDP_1865 := [[11.28, 36.19, 5.43, 0, 48.38, -290.53], [9E9, 9E9, 9E9, 9E9, 9E9, 9E9]];
	VAR jointtarget CDP_1866 := [[11.23, 36.21, 5.39, 0, 48.4, -288.38], [9E9, 9E9, 9E9, 9E9, 9E9, 9E9]];
	VAR jointtarget CDP_1867 := [[11.18, 36.23, 5.36, 0, 48.41, -286.24], [9E9, 9E9, 9E9, 9E9, 9E9, 9E9]];
	VAR jointtarget CDP_1868 := [[11.13, 36.24, 5.34, 0, 48.42, -284.1], [9E9, 9E9, 9E9, 9E9, 9E9, 9E9]];
	VAR jointtarget CDP_1869 := [[11.07, 36.26, 5.32, 0, 48.43, -281.96], [9E9, 9E9, 9E9, 9E9, 9E9, 9E9]];
	VAR jointtarget CDP_1870 := [[11.02, 36.27, 5.3, 0, 48.43, -279.82], [9E9, 9E9, 9E9, 9E9, 9E9, 9E9]];
	VAR jointtarget CDP_1871 := [[10.96, 36.27, 5.29, 0, 48.44, -277.69], [9E9, 9E9, 9E9, 9E9, 9E9, 9E9]];
	VAR jointtarget CDP_1872 := [[10.91, 36.28, 5.28, 0, 48.44, -275.55], [9E9, 9E9, 9E9, 9E9, 9E9, 9E9]];
	VAR jointtarget CDP_1873 := [[10.85, 36.28, 5.27, 0, 48.45, -273.41], [9E9, 9E9, 9E9, 9E9, 9E9, 9E9]];
	VAR jointtarget CDP_1874 := [[10.8, 36.28, 5.27, 0, 48.45, -271.27], [9E9, 9E9, 9E9, 9E9, 9E9, 9E9]];
	VAR jointtarget CDP_1875 := [[10.74, 36.28, 5.27, 0, 48.45, -269.13], [9E9, 9E9, 9E9, 9E9, 9E9, 9E9]];
	VAR jointtarget CDP_1876 := [[10.69, 36.28, 5.27, 0, 48.45, -266.99], [9E9, 9E9, 9E9, 9E9, 9E9, 9E9]];
	VAR jointtarget CDP_1877 := [[10.63, 36.27, 5.28, 0, 48.44, -264.85], [9E9, 9E9, 9E9, 9E9, 9E9, 9E9]];
	VAR jointtarget CDP_1878 := [[10.58, 36.27, 5.3, 0, 48.44, -262.71], [9E9, 9E9, 9E9, 9E9, 9E9, 9E9]];
	VAR jointtarget CDP_1879 := [[10.52, 36.26, 5.31, 0, 48.43, -260.58], [9E9, 9E9, 9E9, 9E9, 9E9, 9E9]];
	VAR jointtarget CDP_1880 := [[9.44, 36.05, 5.67, 0, 48.28, -260.56], [9E9, 9E9, 9E9, 9E9, 9E9, 9E9]];
	VAR jointtarget CDP_1881 := [[8.36, 35.87, 5.98, 0, 48.15, -261.64], [9E9, 9E9, 9E9, 9E9, 9E9, 9E9]];
	VAR jointtarget CDP_1882 := [[7.27, 35.7, 6.26, 0, 48.03, -262.73], [9E9, 9E9, 9E9, 9E9, 9E9, 9E9]];
	VAR jointtarget CDP_1883 := [[6.17, 35.57, 6.5, 0, 47.94, -263.83], [9E9, 9E9, 9E9, 9E9, 9E9, 9E9]];
	VAR jointtarget CDP_1884 := [[5.07, 35.45, 6.7, 0, 47.85, -264.93], [9E9, 9E9, 9E9, 9E9, 9E9, 9E9]];
	VAR jointtarget CDP_1885 := [[3.97, 35.36, 6.86, 0, 47.79, -266.03], [9E9, 9E9, 9E9, 9E9, 9E9, 9E9]];
	VAR jointtarget CDP_1886 := [[2.86, 35.29, 6.98, 0, 47.74, -267.14], [9E9, 9E9, 9E9, 9E9, 9E9, 9E9]];
	VAR jointtarget CDP_1887 := [[1.75, 35.24, 7.06, 0, 47.7, -268.25], [9E9, 9E9, 9E9, 9E9, 9E9, 9E9]];
	VAR jointtarget CDP_1888 := [[0.64, 35.21, 7.1, 0, 47.69, -269.36], [9E9, 9E9, 9E9, 9E9, 9E9, 9E9]];
	VAR jointtarget CDP_1889 := [[-0.47, 35.21, 7.1, 0, 47.68, -270.47], [9E9, 9E9, 9E9, 9E9, 9E9, 9E9]];
	VAR jointtarget CDP_1890 := [[-1.58, 35.23, 7.07, 0, 47.7, -271.58], [9E9, 9E9, 9E9, 9E9, 9E9, 9E9]];
	VAR jointtarget CDP_1891 := [[-2.69, 35.28, 6.99, 0, 47.73, -272.69], [9E9, 9E9, 9E9, 9E9, 9E9, 9E9]];
	VAR jointtarget CDP_1892 := [[-3.8, 35.34, 6.88, 0, 47.78, -273.8], [9E9, 9E9, 9E9, 9E9, 9E9, 9E9]];
	VAR jointtarget CDP_1893 := [[-4.9, 35.43, 6.72, 0, 47.84, -274.9], [9E9, 9E9, 9E9, 9E9, 9E9, 9E9]];
	VAR jointtarget CDP_1894 := [[-6, 35.55, 6.53, 0, 47.92, -276], [9E9, 9E9, 9E9, 9E9, 9E9, 9E9]];
	VAR jointtarget CDP_1895 := [[-7.1, 35.68, 6.3, 0, 48.02, -277.1], [9E9, 9E9, 9E9, 9E9, 9E9, 9E9]];
	VAR jointtarget CDP_1896 := [[-8.19, 35.84, 6.03, 0, 48.13, -278.19], [9E9, 9E9, 9E9, 9E9, 9E9, 9E9]];
	VAR jointtarget CDP_1897 := [[-9.28, 36.02, 5.72, 0, 48.26, -279.28], [9E9, 9E9, 9E9, 9E9, 9E9, 9E9]];
	VAR jointtarget CDP_1898 := [[-10.36, 36.22, 5.37, 0, 48.41, -280.36], [9E9, 9E9, 9E9, 9E9, 9E9, 9E9]];
	VAR jointtarget CDP_1899 := [[-11.43, 36.45, 4.98, 0, 48.57, -281.43], [9E9, 9E9, 9E9, 9E9, 9E9, 9E9]];
	VAR jointtarget CDP_1900 := [[-11.44, 36.45, 4.98, 0, 48.57, -281.78], [9E9, 9E9, 9E9, 9E9, 9E9, 9E9]];
	VAR jointtarget CDP_1901 := [[-11.46, 36.46, 4.97, 0, 48.57, -282.45], [9E9, 9E9, 9E9, 9E9, 9E9, 9E9]];
	VAR jointtarget CDP_1902 := [[-11.48, 36.46, 4.96, 0, 48.58, -283.13], [9E9, 9E9, 9E9, 9E9, 9E9, 9E9]];
	VAR jointtarget CDP_1903 := [[-11.49, 36.47, 4.96, 0, 48.58, -283.81], [9E9, 9E9, 9E9, 9E9, 9E9, 9E9]];
	VAR jointtarget CDP_1904 := [[-11.51, 36.47, 4.95, 0, 48.58, -284.49], [9E9, 9E9, 9E9, 9E9, 9E9, 9E9]];
	VAR jointtarget CDP_1905 := [[-11.53, 36.48, 4.94, 0, 48.59, -285.17], [9E9, 9E9, 9E9, 9E9, 9E9, 9E9]];
	VAR jointtarget CDP_1906 := [[-11.54, 36.48, 4.93, 0, 48.59, -285.84], [9E9, 9E9, 9E9, 9E9, 9E9, 9E9]];
	VAR jointtarget CDP_1907 := [[-11.56, 36.49, 4.92, 0, 48.59, -286.52], [9E9, 9E9, 9E9, 9E9, 9E9, 9E9]];
	VAR jointtarget CDP_1908 := [[-11.57, 36.49, 4.91, 0, 48.6, -287.2], [9E9, 9E9, 9E9, 9E9, 9E9, 9E9]];
	VAR jointtarget CDP_1909 := [[-11.59, 36.5, 4.9, 0, 48.6, -287.88], [9E9, 9E9, 9E9, 9E9, 9E9, 9E9]];
	VAR jointtarget CDP_1910 := [[-11.6, 36.5, 4.89, 0, 48.6, -288.56], [9E9, 9E9, 9E9, 9E9, 9E9, 9E9]];
	VAR jointtarget CDP_1911 := [[-11.62, 36.51, 4.88, 0, 48.61, -289.23], [9E9, 9E9, 9E9, 9E9, 9E9, 9E9]];
	VAR jointtarget CDP_1912 := [[-11.64, 36.51, 4.87, 0, 48.61, -289.91], [9E9, 9E9, 9E9, 9E9, 9E9, 9E9]];
	VAR jointtarget CDP_1913 := [[-11.65, 36.52, 4.86, 0, 48.62, -290.59], [9E9, 9E9, 9E9, 9E9, 9E9, 9E9]];
	VAR jointtarget CDP_1914 := [[-11.67, 36.53, 4.85, 0, 48.62, -291.27], [9E9, 9E9, 9E9, 9E9, 9E9, 9E9]];
	VAR jointtarget CDP_1915 := [[-11.68, 36.53, 4.84, 0, 48.63, -291.94], [9E9, 9E9, 9E9, 9E9, 9E9, 9E9]];
	VAR jointtarget CDP_1916 := [[-11.7, 36.54, 4.83, 0, 48.63, -292.62], [9E9, 9E9, 9E9, 9E9, 9E9, 9E9]];
	VAR jointtarget CDP_1917 := [[-11.71, 36.55, 4.81, 0, 48.64, -293.3], [9E9, 9E9, 9E9, 9E9, 9E9, 9E9]];
	VAR jointtarget CDP_1918 := [[-11.73, 36.56, 4.8, 0, 48.64, -293.98], [9E9, 9E9, 9E9, 9E9, 9E9, 9E9]];
	VAR jointtarget CDP_1919 := [[-11.74, 36.56, 4.79, 0, 48.65, -294.65], [9E9, 9E9, 9E9, 9E9, 9E9, 9E9]];
	VAR jointtarget CDP_1920 := [[-11.8, 36.59, 4.73, 0, 48.67, -295.04], [9E9, 9E9, 9E9, 9E9, 9E9, 9E9]];
	VAR jointtarget CDP_1921 := [[-11.86, 36.63, 4.68, 0, 48.69, -295.11], [9E9, 9E9, 9E9, 9E9, 9E9, 9E9]];
	VAR jointtarget CDP_1922 := [[-11.93, 36.66, 4.63, 0, 48.72, -295.17], [9E9, 9E9, 9E9, 9E9, 9E9, 9E9]];
	VAR jointtarget CDP_1923 := [[-11.99, 36.69, 4.57, 0, 48.74, -295.23], [9E9, 9E9, 9E9, 9E9, 9E9, 9E9]];
	VAR jointtarget CDP_1924 := [[-12.05, 36.72, 4.52, 0, 48.76, -295.29], [9E9, 9E9, 9E9, 9E9, 9E9, 9E9]];
	VAR jointtarget CDP_1925 := [[-12.11, 36.75, 4.46, 0, 48.78, -295.35], [9E9, 9E9, 9E9, 9E9, 9E9, 9E9]];
	VAR jointtarget CDP_1926 := [[-12.17, 36.78, 4.41, 0, 48.81, -295.41], [9E9, 9E9, 9E9, 9E9, 9E9, 9E9]];
	VAR jointtarget CDP_1927 := [[-12.23, 36.82, 4.35, 0, 48.83, -295.47], [9E9, 9E9, 9E9, 9E9, 9E9, 9E9]];
	VAR jointtarget CDP_1928 := [[-12.29, 36.85, 4.3, 0, 48.85, -295.53], [9E9, 9E9, 9E9, 9E9, 9E9, 9E9]];
	VAR jointtarget CDP_1929 := [[-12.35, 36.88, 4.24, 0, 48.88, -295.59], [9E9, 9E9, 9E9, 9E9, 9E9, 9E9]];
	VAR jointtarget CDP_1930 := [[-12.41, 36.91, 4.19, 0, 48.9, -295.65], [9E9, 9E9, 9E9, 9E9, 9E9, 9E9]];
	VAR jointtarget CDP_1931 := [[-12.47, 36.94, 4.13, 0, 48.92, -295.71], [9E9, 9E9, 9E9, 9E9, 9E9, 9E9]];
	VAR jointtarget CDP_1932 := [[-12.53, 36.98, 4.08, 0, 48.95, -295.77], [9E9, 9E9, 9E9, 9E9, 9E9, 9E9]];
	VAR jointtarget CDP_1933 := [[-12.59, 37.01, 4.02, 0, 48.97, -295.83], [9E9, 9E9, 9E9, 9E9, 9E9, 9E9]];
	VAR jointtarget CDP_1934 := [[-12.65, 37.04, 3.97, 0, 48.99, -295.89], [9E9, 9E9, 9E9, 9E9, 9E9, 9E9]];
	VAR jointtarget CDP_1935 := [[-12.71, 37.07, 3.91, 0, 49.02, -295.95], [9E9, 9E9, 9E9, 9E9, 9E9, 9E9]];
	VAR jointtarget CDP_1936 := [[-12.77, 37.1, 3.86, 0, 49.04, -296.01], [9E9, 9E9, 9E9, 9E9, 9E9, 9E9]];
	VAR jointtarget CDP_1937 := [[-12.83, 37.14, 3.8, 0, 49.06, -296.07], [9E9, 9E9, 9E9, 9E9, 9E9, 9E9]];
	VAR jointtarget CDP_1938 := [[-12.89, 37.17, 3.74, 0, 49.09, -296.13], [9E9, 9E9, 9E9, 9E9, 9E9, 9E9]];
	VAR jointtarget CDP_1939 := [[-12.95, 37.2, 3.69, 0, 49.11, -296.19], [9E9, 9E9, 9E9, 9E9, 9E9, 9E9]];
	VAR jointtarget CDP_1940 := [[-13.07, 37.25, 3.6, 0, 49.15, -291.14], [9E9, 9E9, 9E9, 9E9, 9E9, 9E9]];
	VAR jointtarget CDP_1941 := [[-13.19, 37.28, 3.55, 0, 49.17, -280.95], [9E9, 9E9, 9E9, 9E9, 9E9, 9E9]];
	VAR jointtarget CDP_1942 := [[-13.32, 37.28, 3.55, 0, 49.17, -270.75], [9E9, 9E9, 9E9, 9E9, 9E9, 9E9]];
	VAR jointtarget CDP_1943 := [[-13.45, 37.26, 3.59, 0, 49.15, -260.55], [9E9, 9E9, 9E9, 9E9, 9E9, 9E9]];
	VAR jointtarget CDP_1944 := [[-13.57, 37.21, 3.67, 0, 49.12, -250.35], [9E9, 9E9, 9E9, 9E9, 9E9, 9E9]];
	VAR jointtarget CDP_1945 := [[-13.68, 37.14, 3.8, 0, 49.06, -240.14], [9E9, 9E9, 9E9, 9E9, 9E9, 9E9]];
	VAR jointtarget CDP_1946 := [[-13.78, 37.05, 3.96, 0, 49, -229.91], [9E9, 9E9, 9E9, 9E9, 9E9, 9E9]];
	VAR jointtarget CDP_1947 := [[-13.86, 36.94, 4.15, 0, 48.92, -219.67], [9E9, 9E9, 9E9, 9E9, 9E9, 9E9]];
	VAR jointtarget CDP_1948 := [[-13.93, 36.81, 4.36, 0, 48.83, -209.41], [9E9, 9E9, 9E9, 9E9, 9E9, 9E9]];
